LIN {X -0.125,Y -582.899,Z 496.268,A 0.000,B 0.000,C 90.000,E1 264.261} C_DIS
LIN {X -0.140,Y -579.949,Z 496.259,A 0.000,B 0.000,C 90.000,E1 262.648} C_DIS
LIN {X 0.066,Y -576.563,Z 496.249,A 0.000,B 0.000,C 90.000,E1 260.735} C_DIS
LIN {X -0.121,Y -574.110,Z 496.241,A 0.000,B 0.000,C 90.000,E1 259.398} C_DIS
LIN {X -0.046,Y -570.835,Z 496.232,A 0.000,B 0.000,C 90.000,E1 257.757} C_DIS
LIN {X -0.043,Y -567.459,Z 496.223,A 0.000,B 0.000,C 90.000,E1 256.117} C_DIS
LIN {X 0.233,Y -565.087,Z 496.217,A 0.000,B 0.000,C 90.000,E1 254.991} C_DIS
LIN {X -0.069,Y -562.642,Z 496.211,A 0.000,B 0.000,C 90.000,E1 253.921} C_DIS
LIN {X -0.106,Y -559.363,Z 496.203,A 0.000,B 0.000,C 90.000,E1 252.543} C_DIS
LIN {X -0.026,Y -555.962,Z 496.195,A 0.000,B 0.000,C 90.000,E1 251.148} C_DIS
LIN {X 0.080,Y -551.464,Z 496.186,A 0.000,B 0.000,C 90.000,E1 249.464} C_DIS
LIN {X 0.139,Y -548.336,Z 496.180,A 0.000,B 0.000,C 90.000,E1 248.337} C_DIS
LIN {X -0.042,Y -545.121,Z 496.174,A 0.000,B 0.000,C 90.000,E1 247.230} C_DIS
LIN {X -0.059,Y -541.722,Z 496.167,A 0.000,B 0.000,C 90.000,E1 246.102} C_DIS
LIN {X 0.095,Y -537.343,Z 496.159,A 0.000,B 0.000,C 90.000,E1 244.665} C_DIS
LIN {X 0.192,Y -533.762,Z 496.153,A 0.000,B 0.000,C 90.000,E1 243.512} C_DIS
LIN {X 0.238,Y -530.130,Z 496.147,A 0.000,B 0.000,C 90.000,E1 242.359} C_DIS
LIN {X 0.260,Y -523.726,Z 496.135,A 0.000,B 0.000,C 90.000,E1 240.333} C_DIS
LIN {X -0.110,Y -519.148,Z 496.127,A 0.000,B 0.000,C 90.000,E1 238.918} C_DIS
LIN {X -0.043,Y -515.453,Z 496.121,A 0.000,B 0.000,C 90.000,E1 237.740} C_DIS
LIN {X 0.053,Y -509.649,Z 496.111,A 0.000,B 0.000,C 90.000,E1 235.960} C_DIS
LIN {X -0.004,Y -504.726,Z 496.103,A 0.000,B 0.000,C 90.000,E1 234.482} C_DIS
LIN {X 0.032,Y -498.936,Z 496.093,A 0.000,B 0.000,C 90.000,E1 232.683} C_DIS
LIN {X -0.033,Y -489.905,Z 496.076,A 0.000,B 0.000,C 90.000,E1 229.666} C_DIS
LIN {X -0.260,Y -483.929,Z 496.064,A 0.000,B 0.000,C 90.000,E1 227.553} C_DIS
LIN {X 0.082,Y -479.810,Z 496.056,A 0.000,B 0.000,C 90.000,E1 225.972} C_DIS
LIN {X 0.215,Y -474.180,Z 496.043,A 0.000,B 0.000,C 90.000,E1 223.785} C_DIS
LIN {X 0.047,Y -470.290,Z 496.035,A 0.000,B 0.000,C 90.000,E1 222.243} C_DIS
LIN {X -0.124,Y -465.832,Z 496.024,A 0.000,B 0.000,C 90.000,E1 220.378} C_DIS
LIN {X -0.245,Y -460.903,Z 496.012,A 0.000,B 0.000,C 90.000,E1 218.177} C_DIS
LIN {X -0.034,Y -455.639,Z 495.998,A 0.000,B 0.000,C 90.000,E1 215.598} C_DIS
LIN {X 0.057,Y -451.793,Z 495.987,A 0.000,B 0.000,C 90.000,E1 213.658} C_DIS
LIN {X 0.051,Y -448.147,Z 495.976,A 0.000,B 0.000,C 90.000,E1 211.720} C_DIS
LIN {X -0.203,Y -445.158,Z 495.967,A 0.000,B 0.000,C 90.000,E1 210.129} C_DIS
LIN {X -0.235,Y -441.032,Z 495.955,A 0.000,B 0.000,C 90.000,E1 207.847} C_DIS
LIN {X -0.049,Y -438.068,Z 495.945,A 0.000,B 0.000,C 90.000,E1 206.181} C_DIS
LIN {X 0.060,Y -435.744,Z 495.938,A 0.000,B 0.000,C 90.000,E1 204.847} C_DIS
LIN {X -0.228,Y -432.280,Z 495.927,A 0.000,B 0.000,C 90.000,E1 202.898} C_DIS
LIN {X -0.159,Y -428.358,Z 495.914,A 0.000,B 0.000,C 90.000,E1 200.556} C_DIS
LIN {X -0.143,Y -425.321,Z 495.903,A 0.000,B 0.000,C 90.000,E1 198.544} C_DIS
LIN {X 0.128,Y -420.629,Z 495.884,A 0.000,B 0.000,C 90.000,E1 195.134} C_DIS
LIN {X 0.042,Y -417.671,Z 495.871,A 0.000,B 0.000,C 90.000,E1 192.771} C_DIS
LIN {X -0.001,Y -415.716,Z 495.862,A 0.000,B 0.000,C 90.000,E1 191.074} C_DIS
LIN {X -0.048,Y -413.433,Z 495.850,A 0.000,B 0.000,C 90.000,E1 189.029} C_DIS
LIN {X 0.132,Y -410.700,Z 495.835,A 0.000,B 0.000,C 90.000,E1 186.258} C_DIS
LIN {X 0.162,Y -408.347,Z 495.822,A 0.000,B 0.000,C 90.000,E1 183.841} C_DIS
LIN {X 0.002,Y -405.676,Z 495.802,A 0.000,B 0.000,C 90.000,E1 180.401} C_DIS
LIN {X 0.173,Y -403.932,Z 495.785,A 0.000,B 0.000,C 90.000,E1 177.249} C_DIS
LIN {X -0.065,Y -402.940,Z 495.766,A 0.000,B 0.000,C 90.000,E1 173.799} C_DIS
LIN {X -0.189,Y -402.803,Z 495.754,A 0.000,B 0.000,C 90.000,E1 171.724} C_DIS
LIN {X -0.134,Y -403.045,Z 495.738,A 0.000,B 0.000,C 90.000,E1 168.926} C_DIS
LIN {X 0.015,Y -403.828,Z 495.723,A 0.000,B 0.000,C 90.000,E1 166.117} C_DIS
LIN {X 0.083,Y -404.981,Z 495.707,A 0.000,B 0.000,C 90.000,E1 163.323} C_DIS
LIN {X 0.042,Y -406.645,Z 495.692,A 0.000,B 0.000,C 90.000,E1 160.550} C_DIS
LIN {X 0.212,Y -409.001,Z 495.675,A 0.000,B 0.000,C 90.000,E1 157.411} C_DIS
LIN {X 0.099,Y -410.828,Z 495.663,A 0.000,B 0.000,C 90.000,E1 155.357} C_DIS
LIN {X 0.000,Y -412.786,Z 495.652,A 0.000,B 0.000,C 90.000,E1 153.307} C_DIS
LIN {X 0.009,Y -414.381,Z 495.642,A 0.000,B 0.000,C 90.000,E1 151.591} C_DIS
LIN {X 0.073,Y -415.964,Z 495.633,A 0.000,B 0.000,C 90.000,E1 149.871} C_DIS
LIN {X -0.238,Y -417.734,Z 495.621,A 0.000,B 0.000,C 90.000,E1 147.867} C_DIS
LIN {X -0.200,Y -418.862,Z 495.614,A 0.000,B 0.000,C 90.000,E1 146.501} C_DIS
LIN {X 0.046,Y -420.250,Z 495.604,A 0.000,B 0.000,C 90.000,E1 144.769} C_DIS
LIN {X 0.054,Y -422.224,Z 495.591,A 0.000,B 0.000,C 90.000,E1 142.396} C_DIS
LIN {X 0.158,Y -423.798,Z 495.580,A 0.000,B 0.000,C 90.000,E1 140.356} C_DIS
LIN {X 0.115,Y -424.813,Z 495.572,A 0.000,B 0.000,C 90.000,E1 139.013} C_DIS
LIN {X 0.051,Y -425.666,Z 495.565,A 0.000,B 0.000,C 90.000,E1 137.676} C_DIS
LIN {X 0.093,Y -426.178,Z 495.559,A 0.000,B 0.000,C 90.000,E1 136.662} C_DIS
LIN {X 0.053,Y -426.740,Z 495.552,A 0.000,B 0.000,C 90.000,E1 135.324} C_DIS
LIN {X -0.285,Y -427.019,Z 495.544,A 0.000,B 0.000,C 90.000,E1 134.028} C_DIS
LIN {X 0.148,Y -427.105,Z 495.541,A 0.000,B 0.000,C 90.000,E1 133.299} C_DIS
LIN {X -0.085,Y -426.928,Z 495.535,A 0.000,B 0.000,C 90.000,E1 132.324} C_DIS
LIN {X -0.120,Y -426.340,Z 495.528,A 0.000,B 0.000,C 90.000,E1 130.987} C_DIS
LIN {X -0.029,Y -425.591,Z 495.522,A 0.000,B 0.000,C 90.000,E1 129.967} C_DIS
LIN {X -0.043,Y -424.318,Z 495.515,A 0.000,B 0.000,C 90.000,E1 128.624} C_DIS
LIN {X -0.088,Y -422.876,Z 495.507,A 0.000,B 0.000,C 90.000,E1 127.282} C_DIS
LIN {X -0.081,Y -421.282,Z 495.500,A 0.000,B 0.000,C 90.000,E1 125.931} C_DIS
LIN {X 0.004,Y -419.535,Z 495.492,A 0.000,B 0.000,C 90.000,E1 124.565} C_DIS
LIN {X -0.110,Y -419.290,Z 495.491,A 0.000,B 0.000,C 90.000,E1 124.405} C_DIS
LIN {X -0.148,Y -419.282,Z 495.491,A 0.000,B 0.000,C 90.000,E1 124.405} C_DIS
LIN {X 0.029,Y -429.026,Z 495.471,A 0.000,B 0.000,C 90.000,E1 120.846} C_DIS
LIN {X -0.198,Y -431.019,Z 495.468,A 0.000,B 0.000,C 90.000,E1 120.207} C_DIS
LIN {X -0.054,Y -440.094,Z 495.447,A 0.000,B 0.000,C 90.000,E1 116.539} C_DIS
LIN {X -0.056,Y -444.873,Z 495.438,A 0.000,B 0.000,C 90.000,E1 114.899} C_DIS
LIN {X 0.203,Y -453.984,Z 495.417,A 0.000,B 0.000,C 90.000,E1 110.972} C_DIS
LIN {X -0.270,Y -456.632,Z 495.411,A 0.000,B 0.000,C 90.000,E1 110.066} C_DIS
LIN {X 0.061,Y -457.448,Z 495.410,A 0.000,B 0.000,C 90.000,E1 109.704} C_DIS
LIN {X -0.005,Y -464.473,Z 495.390,A 0.000,B 0.000,C 90.000,E1 106.260} C_DIS
LIN {X -0.045,Y -464.485,Z 495.390,A 0.000,B 0.000,C 90.000,E1 106.260} C_DIS
LIN {X 0.015,Y -471.360,Z 495.390,A 0.000,B 0.000,C 90.000,E1 106.134} C_DIS
LIN {X -0.014,Y -475.196,Z 495.389,A 0.000,B 0.000,C 90.000,E1 106.079} C_DIS
LIN {X -0.202,Y -485.320,Z 495.388,A 0.000,B 0.000,C 90.000,E1 105.898} C_DIS
LIN {X 0.014,Y -492.601,Z 495.387,A 0.000,B 0.000,C 90.000,E1 105.717} C_DIS
LIN {X 0.107,Y -506.770,Z 495.385,A 0.000,B 0.000,C 90.000,E1 105.371} C_DIS
LIN {X -0.249,Y -517.096,Z 495.384,A 0.000,B 0.000,C 90.000,E1 105.134} C_DIS
LIN {X -0.215,Y -527.592,Z 495.382,A 0.000,B 0.000,C 90.000,E1 104.828} C_DIS
LIN {X 0.032,Y -537.871,Z 495.381,A 0.000,B 0.000,C 90.000,E1 104.481} C_DIS
LIN {X 0.104,Y -544.566,Z 495.379,A 0.000,B 0.000,C 90.000,E1 104.245} C_DIS
LIN {X -0.050,Y -551.197,Z 495.378,A 0.000,B 0.000,C 90.000,E1 104.008} C_DIS
LIN {X -0.155,Y -554.500,Z 495.377,A 0.000,B 0.000,C 90.000,E1 103.883} C_DIS
LIN {X 0.048,Y -564.165,Z 495.375,A 0.000,B 0.000,C 90.000,E1 103.411} C_DIS
LIN {X 0.216,Y -567.305,Z 495.374,A 0.000,B 0.000,C 90.000,E1 103.244} C_DIS
LIN {X -0.224,Y -576.586,Z 495.371,A 0.000,B 0.000,C 90.000,E1 102.771} C_DIS
LIN {X 0.092,Y -582.403,Z 495.369,A 0.000,B 0.000,C 90.000,E1 102.355} C_DIS
LIN {X 0.026,Y -586.631,Z 495.367,A 0.000,B 0.000,C 90.000,E1 102.063} C_DIS
LIN {X 0.092,Y -588.353,Z 495.366,A 0.000,B 0.000,C 90.000,E1 101.951} C_DIS
LIN {X 0.279,Y -596.480,Z 495.363,A 0.000,B 0.000,C 90.000,E1 101.299} C_DIS
LIN {X 0.316,Y -600.049,Z 495.361,A 0.000,B 0.000,C 90.000,E1 101.007} C_DIS
LIN {X 0.142,Y -606.738,Z 495.358,A 0.000,B 0.000,C 90.000,E1 100.433} C_DIS
LIN {X -0.193,Y -612.950,Z 495.355,A 0.000,B 0.000,C 90.000,E1 99.849} C_DIS
LIN {X 0.032,Y -617.750,Z 495.352,A 0.000,B 0.000,C 90.000,E1 99.321} C_DIS
LIN {X 0.023,Y -623.315,Z 495.348,A 0.000,B 0.000,C 90.000,E1 98.681} C_DIS
LIN {X 0.098,Y -627.427,Z 495.345,A 0.000,B 0.000,C 90.000,E1 98.163} C_DIS
LIN {X 0.060,Y -632.061,Z 495.342,A 0.000,B 0.000,C 90.000,E1 97.530} C_DIS
LIN {X 0.005,Y -636.964,Z 495.338,A 0.000,B 0.000,C 90.000,E1 96.777} C_DIS
LIN {X 0.180,Y -639.953,Z 495.335,A 0.000,B 0.000,C 90.000,E1 96.258} C_DIS
LIN {X 0.171,Y -644.017,Z 495.331,A 0.000,B 0.000,C 90.000,E1 95.511} C_DIS
LIN {X 0.103,Y -648.345,Z 495.326,A 0.000,B 0.000,C 90.000,E1 94.645} C_DIS
LIN {X 0.303,Y -650.663,Z 495.323,A 0.000,B 0.000,C 90.000,E1 94.131} C_DIS
LIN {X -0.296,Y -653.703,Z 495.319,A 0.000,B 0.000,C 90.000,E1 93.440} C_DIS
LIN {X -0.018,Y -655.493,Z 495.316,A 0.000,B 0.000,C 90.000,E1 92.922} C_DIS
LIN {X 0.240,Y -657.038,Z 495.314,A 0.000,B 0.000,C 90.000,E1 92.407} C_DIS
LIN {X -0.312,Y -658.803,Z 495.309,A 0.000,B 0.000,C 90.000,E1 91.718} C_DIS
LIN {X -0.028,Y -659.700,Z 495.307,A 0.000,B 0.000,C 90.000,E1 91.203} C_DIS
LIN {X 0.265,Y -660.274,Z 495.304,A 0.000,B 0.000,C 90.000,E1 90.688} C_DIS
LIN {X -0.275,Y -660.761,Z 495.300,A 0.000,B 0.000,C 90.000,E1 90.000} C_DIS
LIN {X 0.029,Y -660.764,Z 495.297,A 0.000,B 0.000,C 90.000,E1 89.484} C_DIS
LIN {X 0.151,Y -660.208,Z 495.293,A 0.000,B 0.000,C 90.000,E1 88.740} C_DIS
LIN {X -0.212,Y -659.627,Z 495.290,A 0.000,B 0.000,C 90.000,E1 88.282} C_DIS
LIN {X 0.103,Y -658.852,Z 495.288,A 0.000,B 0.000,C 90.000,E1 87.764} C_DIS
LIN {X -0.268,Y -657.826,Z 495.285,A 0.000,B 0.000,C 90.000,E1 87.306} C_DIS
LIN {X -0.148,Y -655.795,Z 495.281,A 0.000,B 0.000,C 90.000,E1 86.560} C_DIS
LIN {X 0.111,Y -654.200,Z 495.278,A 0.000,B 0.000,C 90.000,E1 86.045} C_DIS
LIN {X -0.249,Y -652.384,Z 495.275,A 0.000,B 0.000,C 90.000,E1 85.584} C_DIS
LIN {X 0.034,Y -650.350,Z 495.273,A 0.000,B 0.000,C 90.000,E1 85.065} C_DIS
LIN {X 0.081,Y -646.848,Z 495.269,A 0.000,B 0.000,C 90.000,E1 84.318} C_DIS
LIN {X 0.205,Y -643.584,Z 495.265,A 0.000,B 0.000,C 90.000,E1 83.685} C_DIS
LIN {X -0.339,Y -640.018,Z 495.262,A 0.000,B 0.000,C 90.000,E1 83.109} C_DIS
LIN {X -0.197,Y -636.089,Z 495.258,A 0.000,B 0.000,C 90.000,E1 82.470} C_DIS
LIN {X -0.169,Y -631.793,Z 495.255,A 0.000,B 0.000,C 90.000,E1 81.837} C_DIS
LIN {X -0.036,Y -628.041,Z 495.252,A 0.000,B 0.000,C 90.000,E1 81.319} C_DIS
LIN {X 0.054,Y -622.961,Z 495.248,A 0.000,B 0.000,C 90.000,E1 80.679} C_DIS
LIN {X 0.135,Y -617.609,Z 495.245,A 0.000,B 0.000,C 90.000,E1 80.038} C_DIS
LIN {X 0.094,Y -611.756,Z 495.241,A 0.000,B 0.000,C 90.000,E1 79.398} C_DIS
LIN {X 0.139,Y -605.468,Z 495.238,A 0.000,B 0.000,C 90.000,E1 78.757} C_DIS
LIN {X -0.032,Y -600.385,Z 495.235,A 0.000,B 0.000,C 90.000,E1 78.285} C_DIS
LIN {X -0.205,Y -596.393,Z 495.233,A 0.000,B 0.000,C 90.000,E1 77.937} C_DIS
LIN {X -0.068,Y -590.433,Z 495.230,A 0.000,B 0.000,C 90.000,E1 77.465} C_DIS
LIN {X 0.344,Y -584.507,Z 495.228,A 0.000,B 0.000,C 90.000,E1 76.992} C_DIS
LIN {X -0.283,Y -578.256,Z 495.226,A 0.000,B 0.000,C 90.000,E1 76.645} C_DIS
LIN {X -0.252,Y -573.325,Z 495.224,A 0.000,B 0.000,C 90.000,E1 76.353} C_DIS
LIN {X -0.124,Y -566.598,Z 495.222,A 0.000,B 0.000,C 90.000,E1 75.992} C_DIS
LIN {X -0.266,Y -559.098,Z 495.220,A 0.000,B 0.000,C 90.000,E1 75.700} C_DIS
LIN {X 0.117,Y -555.118,Z 495.220,A 0.000,B 0.000,C 90.000,E1 75.519} C_DIS
LIN {X 0.209,Y -547.325,Z 495.218,A 0.000,B 0.000,C 90.000,E1 75.283} C_DIS
LIN {X -0.047,Y -540.716,Z 495.218,A 0.000,B 0.000,C 90.000,E1 75.172} C_DIS
LIN {X 0.174,Y -534.917,Z 495.217,A 0.000,B 0.000,C 90.000,E1 75.046} C_DIS
LIN {X -0.132,Y -527.738,Z 495.217,A 0.000,B 0.000,C 90.000,E1 74.991} C_DIS
LIN {X -0.034,Y -523.125,Z 495.216,A 0.000,B 0.000,C 90.000,E1 74.936} C_DIS
LIN {X 0.189,Y -512.995,Z 495.216,A 0.000,B 0.000,C 90.000,E1 74.866} C_DIS
LIN {X -0.025,Y -504.486,Z 495.216,A 0.000,B 0.000,C 90.000,E1 74.866} C_DIS
LIN {X -0.053,Y -477.448,Z 495.216,A 0.000,B 0.000,C 90.000,E1 74.866} C_DIS
LIN {X 0.011,Y -474.312,Z 495.201,A 0.000,B 0.000,C 90.000,E1 72.236} C_DIS
LIN {X -0.168,Y -473.904,Z 495.200,A 0.000,B 0.000,C 90.000,E1 71.945} C_DIS
LIN {X -0.041,Y -466.293,Z 495.175,A 0.000,B 0.000,C 90.000,E1 67.539} C_DIS
LIN {X -0.099,Y -465.863,Z 495.173,A 0.000,B 0.000,C 90.000,E1 67.230} C_DIS
LIN {X -0.157,Y -465.298,Z 495.172,A 0.000,B 0.000,C 90.000,E1 66.922} C_DIS
LIN {X 0.220,Y -456.907,Z 495.149,A 0.000,B 0.000,C 90.000,E1 62.743} C_DIS
LIN {X -0.076,Y -455.278,Z 495.143,A 0.000,B 0.000,C 90.000,E1 61.820} C_DIS
LIN {X -0.221,Y -450.847,Z 495.133,A 0.000,B 0.000,C 90.000,E1 59.999} C_DIS
LIN {X 0.130,Y -450.870,Z 495.133,A 0.000,B 0.000,C 90.000,E1 59.950} C_DIS
LIN {X -0.043,Y -456.053,Z 495.127,A 0.000,B 0.000,C 90.000,E1 58.918} C_DIS
LIN {X 0.049,Y -460.472,Z 495.122,A 0.000,B 0.000,C 90.000,E1 57.946} C_DIS
LIN {X -0.097,Y -463.771,Z 495.118,A 0.000,B 0.000,C 90.000,E1 57.168} C_DIS
LIN {X -0.074,Y -466.800,Z 495.113,A 0.000,B 0.000,C 90.000,E1 56.373} C_DIS
LIN {X 0.091,Y -468.866,Z 495.110,A 0.000,B 0.000,C 90.000,E1 55.722} C_DIS
LIN {X 0.170,Y -471.543,Z 495.104,A 0.000,B 0.000,C 90.000,E1 54.769} C_DIS
LIN {X 0.166,Y -473.662,Z 495.099,A 0.000,B 0.000,C 90.000,E1 53.829} C_DIS
LIN {X 0.118,Y -474.920,Z 495.096,A 0.000,B 0.000,C 90.000,E1 53.210} C_DIS
LIN {X -0.052,Y -476.778,Z 495.089,A 0.000,B 0.000,C 90.000,E1 51.984} C_DIS
LIN {X -0.165,Y -477.602,Z 495.085,A 0.000,B 0.000,C 90.000,E1 51.376} C_DIS
LIN {X -0.098,Y -478.550,Z 495.080,A 0.000,B 0.000,C 90.000,E1 50.436} C_DIS
LIN {X 0.196,Y -479.882,Z 495.072,A 0.000,B 0.000,C 90.000,E1 48.852} C_DIS
LIN {X 0.031,Y -480.562,Z 495.065,A 0.000,B 0.000,C 90.000,E1 47.634} C_DIS
LIN {X 0.074,Y -480.980,Z 495.060,A 0.000,B 0.000,C 90.000,E1 46.701} C_DIS
LIN {X -0.227,Y -481.214,Z 495.054,A 0.000,B 0.000,C 90.000,E1 45.810} C_DIS
LIN {X -0.056,Y -481.357,Z 495.048,A 0.000,B 0.000,C 90.000,E1 44.555} C_DIS
LIN {X 0.120,Y -481.316,Z 495.041,A 0.000,B 0.000,C 90.000,E1 43.299} C_DIS
LIN {X -0.028,Y -480.996,Z 495.034,A 0.000,B 0.000,C 90.000,E1 42.081} C_DIS
LIN {X 0.142,Y -480.437,Z 495.027,A 0.000,B 0.000,C 90.000,E1 40.825} C_DIS
LIN {X -0.042,Y -479.466,Z 495.017,A 0.000,B 0.000,C 90.000,E1 38.991} C_DIS
LIN {X -0.241,Y -478.407,Z 495.006,A 0.000,B 0.000,C 90.000,E1 37.156} C_DIS
LIN {X -0.176,Y -477.402,Z 494.998,A 0.000,B 0.000,C 90.000,E1 35.598} C_DIS
LIN {X 0.050,Y -475.869,Z 494.987,A 0.000,B 0.000,C 90.000,E1 33.706} C_DIS
LIN {X -0.001,Y -474.826,Z 494.980,A 0.000,B 0.000,C 90.000,E1 32.467} C_DIS
LIN {X -0.141,Y -473.414,Z 494.972,A 0.000,B 0.000,C 90.000,E1 30.924} C_DIS
LIN {X 0.097,Y -471.814,Z 494.963,A 0.000,B 0.000,C 90.000,E1 29.333} C_DIS
LIN {X -0.090,Y -470.583,Z 494.956,A 0.000,B 0.000,C 90.000,E1 28.103} C_DIS
LIN {X -0.098,Y -468.318,Z 494.942,A 0.000,B 0.000,C 90.000,E1 25.591} C_DIS
LIN {X -0.275,Y -465.857,Z 494.925,A 0.000,B 0.000,C 90.000,E1 22.461} C_DIS
LIN {X 0.104,Y -464.382,Z 494.911,A 0.000,B 0.000,C 90.000,E1 19.885} C_DIS
LIN {X -0.021,Y -463.424,Z 494.900,A 0.000,B 0.000,C 90.000,E1 18.000} C_DIS
LIN {X -0.088,Y -462.455,Z 494.888,A 0.000,B 0.000,C 90.000,E1 15.788} C_DIS
LIN {X 0.070,Y -461.536,Z 494.870,A 0.000,B 0.000,C 90.000,E1 12.591} C_DIS
LIN {X -0.121,Y -461.260,Z 494.852,A 0.000,B 0.000,C 90.000,E1 9.434} C_DIS
LIN {X -0.130,Y -461.578,Z 494.838,A 0.000,B 0.000,C 90.000,E1 6.891} C_DIS
LIN {X -0.035,Y -462.931,Z 494.819,A 0.000,B 0.000,C 90.000,E1 3.383} C_DIS
LIN {X -0.139,Y -464.512,Z 494.805,A 0.000,B 0.000,C 90.000,E1 0.859} C_DIS
LIN {X 0.142,Y -466.475,Z 494.792,A 0.000,B 0.000,C 90.000,E1 358.511} C_DIS
LIN {X -0.081,Y -468.797,Z 494.780,A 0.000,B 0.000,C 90.000,E1 356.331} C_DIS
LIN {X -0.209,Y -471.421,Z 494.767,A 0.000,B 0.000,C 90.000,E1 354.147} C_DIS
LIN {X 0.180,Y -473.420,Z 494.759,A 0.000,B 0.000,C 90.000,E1 352.534} C_DIS
LIN {X -0.128,Y -476.341,Z 494.747,A 0.000,B 0.000,C 90.000,E1 350.387} C_DIS
LIN {X 0.200,Y -479.684,Z 494.734,A 0.000,B 0.000,C 90.000,E1 348.173} C_DIS
LIN {X 0.222,Y -484.142,Z 494.721,A 0.000,B 0.000,C 90.000,E1 345.700} C_DIS
LIN {X 0.157,Y -488.504,Z 494.709,A 0.000,B 0.000,C 90.000,E1 343.559} C_DIS
LIN {X -0.033,Y -491.770,Z 494.700,A 0.000,B 0.000,C 90.000,E1 342.054} C_DIS
LIN {X -0.070,Y -496.463,Z 494.689,A 0.000,B 0.000,C 90.000,E1 339.934} C_DIS
LIN {X 0.045,Y -499.848,Z 494.680,A 0.000,B 0.000,C 90.000,E1 338.411} C_DIS
LIN {X -0.061,Y -503.163,Z 494.672,A 0.000,B 0.000,C 90.000,E1 336.922} C_DIS
LIN {X 0.096,Y -506.347,Z 494.663,A 0.000,B 0.000,C 90.000,E1 335.409} C_DIS
LIN {X -0.142,Y -509.441,Z 494.655,A 0.000,B 0.000,C 90.000,E1 333.948} C_DIS
LIN {X 0.009,Y -513.160,Z 494.645,A 0.000,B 0.000,C 90.000,E1 332.153} C_DIS
LIN {X 0.136,Y -517.602,Z 494.634,A 0.000,B 0.000,C 90.000,E1 330.078} C_DIS
LIN {X 0.110,Y -522.861,Z 494.621,A 0.000,B 0.000,C 90.000,E1 327.740} C_DIS
LIN {X -0.038,Y -527.524,Z 494.610,A 0.000,B 0.000,C 90.000,E1 325.722} C_DIS
LIN {X -0.047,Y -531.597,Z 494.600,A 0.000,B 0.000,C 90.000,E1 323.989} C_DIS
LIN {X -0.093,Y -535.702,Z 494.590,A 0.000,B 0.000,C 90.000,E1 322.271} C_DIS
LIN {X 0.267,Y -539.018,Z 494.582,A 0.000,B 0.000,C 90.000,E1 320.803} C_DIS
LIN {X 0.275,Y -542.391,Z 494.575,A 0.000,B 0.000,C 90.000,E1 319.380} C_DIS
LIN {X -0.068,Y -545.702,Z 494.567,A 0.000,B 0.000,C 90.000,E1 318.000} C_DIS
LIN {X 0.018,Y -548.934,Z 494.559,A 0.000,B 0.000,C 90.000,E1 316.581} C_DIS
LIN {X 0.162,Y -552.044,Z 494.551,A 0.000,B 0.000,C 90.000,E1 315.162} C_DIS
LIN {X 0.016,Y -555.740,Z 494.542,A 0.000,B 0.000,C 90.000,E1 313.500} C_DIS
LIN {X -0.054,Y -559.395,Z 494.532,A 0.000,B 0.000,C 90.000,E1 311.838} C_DIS
LIN {X -0.103,Y -562.458,Z 494.525,A 0.000,B 0.000,C 90.000,E1 310.458} C_DIS
LIN {X -0.360,Y -566.015,Z 494.516,A 0.000,B 0.000,C 90.000,E1 308.830} C_DIS
LIN {X 0.029,Y -570.242,Z 494.505,A 0.000,B 0.000,C 90.000,E1 306.870} C_DIS
LIN {X 0.177,Y -574.605,Z 494.494,A 0.000,B 0.000,C 90.000,E1 304.945} C_DIS
LIN {X 0.265,Y -577.718,Z 494.487,A 0.000,B 0.000,C 90.000,E1 303.579} C_DIS
LIN {X -0.068,Y -582.051,Z 494.476,A 0.000,B 0.000,C 90.000,E1 301.720} C_DIS
LIN {X -0.161,Y -584.832,Z 494.469,A 0.000,B 0.000,C 90.000,E1 300.384} C_DIS
LIN {X 0.134,Y -586.980,Z 494.463,A 0.000,B 0.000,C 90.000,E1 299.283} C_DIS
LIN {X -0.048,Y -588.958,Z 494.457,A 0.000,B 0.000,C 90.000,E1 298.231} C_DIS
LIN {X -0.103,Y -590.292,Z 494.452,A 0.000,B 0.000,C 90.000,E1 297.436} C_DIS
LIN {X 0.004,Y -591.878,Z 494.447,A 0.000,B 0.000,C 90.000,E1 296.360} C_DIS
LIN {X 0.143,Y -593.252,Z 494.441,A 0.000,B 0.000,C 90.000,E1 295.283} C_DIS
LIN {X 0.302,Y -594.387,Z 494.435,A 0.000,B 0.000,C 90.000,E1 294.207} C_DIS
LIN {X -0.313,Y -595.281,Z 494.429,A 0.000,B 0.000,C 90.000,E1 293.206} C_DIS
LIN {X -0.004,Y -596.457,Z 494.420,A 0.000,B 0.000,C 90.000,E1 291.589} C_DIS
LIN {X -0.261,Y -597.158,Z 494.414,A 0.000,B 0.000,C 90.000,E1 290.556} C_DIS
LIN {X 0.263,Y -597.722,Z 494.408,A 0.000,B 0.000,C 90.000,E1 289.450} C_DIS
LIN {X -0.103,Y -598.445,Z 494.398,A 0.000,B 0.000,C 90.000,E1 287.638} C_DIS
LIN {X -0.225,Y -598.739,Z 494.394,A 0.000,B 0.000,C 90.000,E1 286.858} C_DIS
LIN {X 0.110,Y -599.251,Z 494.385,A 0.000,B 0.000,C 90.000,E1 285.245} C_DIS
LIN {X -0.003,Y -599.587,Z 494.377,A 0.000,B 0.000,C 90.000,E1 283.939} C_DIS
LIN {X -0.257,Y -599.822,Z 494.370,A 0.000,B 0.000,C 90.000,E1 282.647} C_DIS
LIN {X 0.078,Y -599.922,Z 494.363,A 0.000,B 0.000,C 90.000,E1 281.299} C_DIS
LIN {X 0.302,Y -599.890,Z 494.356,A 0.000,B 0.000,C 90.000,E1 279.962} C_DIS
LIN {X -0.070,Y -599.713,Z 494.348,A 0.000,B 0.000,C 90.000,E1 278.681} C_DIS
LIN {X 0.057,Y -599.361,Z 494.341,A 0.000,B 0.000,C 90.000,E1 277.352} C_DIS
LIN {X -0.111,Y -598.977,Z 494.335,A 0.000,B 0.000,C 90.000,E1 276.315} C_DIS
LIN {X -0.058,Y -598.209,Z 494.328,A 0.000,B 0.000,C 90.000,E1 274.992} C_DIS
LIN {X -0.019,Y -597.189,Z 494.320,A 0.000,B 0.000,C 90.000,E1 273.669} C_DIS
LIN {X -0.037,Y -596.002,Z 494.313,A 0.000,B 0.000,C 90.000,E1 272.350} C_DIS
LIN {X -0.078,Y -594.463,Z 494.306,A 0.000,B 0.000,C 90.000,E1 271.031} C_DIS
LIN {X -0.158,Y -592.713,Z 494.298,A 0.000,B 0.000,C 90.000,E1 269.714} C_DIS
LIN {X -0.273,Y -590.819,Z 494.291,A 0.000,B 0.000,C 90.000,E1 268.396} C_DIS
LIN {X -0.176,Y -588.465,Z 494.282,A 0.000,B 0.000,C 90.000,E1 266.788} C_DIS
LIN {X 0.237,Y -586.364,Z 494.275,A 0.000,B 0.000,C 90.000,E1 265.412} C_DIS
LIN {X -0.108,Y -584.532,Z 494.269,A 0.000,B 0.000,C 90.000,E1 264.375} C_DIS
LIN {X -0.312,Y -582.002,Z 494.261,A 0.000,B 0.000,C 90.000,E1 263.053} C_DIS
LIN {X 0.161,Y -579.504,Z 494.254,A 0.000,B 0.000,C 90.000,E1 261.659} C_DIS
LIN {X 0.148,Y -576.576,Z 494.245,A 0.000,B 0.000,C 90.000,E1 260.038} C_DIS
LIN {X -0.044,Y -573.904,Z 494.237,A 0.000,B 0.000,C 90.000,E1 258.701} C_DIS
LIN {X -0.172,Y -571.088,Z 494.230,A 0.000,B 0.000,C 90.000,E1 257.353} C_DIS
LIN {X -0.215,Y -568.227,Z 494.222,A 0.000,B 0.000,C 90.000,E1 255.992} C_DIS
LIN {X -0.138,Y -564.549,Z 494.213,A 0.000,B 0.000,C 90.000,E1 254.338} C_DIS
LIN {X -0.140,Y -561.268,Z 494.205,A 0.000,B 0.000,C 90.000,E1 252.960} C_DIS
LIN {X -0.202,Y -557.856,Z 494.198,A 0.000,B 0.000,C 90.000,E1 251.583} C_DIS
LIN {X 0.269,Y -554.949,Z 494.191,A 0.000,B 0.000,C 90.000,E1 250.423} C_DIS
LIN {X -0.015,Y -551.875,Z 494.185,A 0.000,B 0.000,C 90.000,E1 249.337} C_DIS
LIN {X -0.149,Y -548.743,Z 494.179,A 0.000,B 0.000,C 90.000,E1 248.230} C_DIS
LIN {X -0.119,Y -545.436,Z 494.173,A 0.000,B 0.000,C 90.000,E1 247.102} C_DIS
LIN {X 0.126,Y -542.890,Z 494.168,A 0.000,B 0.000,C 90.000,E1 246.230} C_DIS
LIN {X 0.077,Y -539.350,Z 494.162,A 0.000,B 0.000,C 90.000,E1 245.101} C_DIS
LIN {X -0.069,Y -534.880,Z 494.154,A 0.000,B 0.000,C 90.000,E1 243.691} C_DIS
LIN {X 0.181,Y -530.290,Z 494.146,A 0.000,B 0.000,C 90.000,E1 242.231} C_DIS
LIN {X 0.207,Y -523.855,Z 494.135,A 0.000,B 0.000,C 90.000,E1 240.205} C_DIS
LIN {X -0.164,Y -519.244,Z 494.127,A 0.000,B 0.000,C 90.000,E1 238.791} C_DIS
LIN {X 0.179,Y -515.530,Z 494.120,A 0.000,B 0.000,C 90.000,E1 237.582} C_DIS
LIN {X 0.284,Y -509.685,Z 494.110,A 0.000,B 0.000,C 90.000,E1 235.801} C_DIS
LIN {X -0.063,Y -504.725,Z 494.102,A 0.000,B 0.000,C 90.000,E1 234.356} C_DIS
LIN {X -0.033,Y -498.915,Z 494.092,A 0.000,B 0.000,C 90.000,E1 232.557} C_DIS
LIN {X 0.048,Y -490.779,Z 494.077,A 0.000,B 0.000,C 90.000,E1 229.828} C_DIS
LIN {X 0.019,Y -485.592,Z 494.067,A 0.000,B 0.000,C 90.000,E1 228.000} C_DIS
LIN {X 0.064,Y -481.441,Z 494.058,A 0.000,B 0.000,C 90.000,E1 226.458} C_DIS
LIN {X -0.322,Y -474.926,Z 494.044,A 0.000,B 0.000,C 90.000,E1 224.028} C_DIS
LIN {X -0.154,Y -471.027,Z 494.036,A 0.000,B 0.000,C 90.000,E1 222.447} C_DIS
LIN {X 0.041,Y -466.546,Z 494.025,A 0.000,B 0.000,C 90.000,E1 220.539} C_DIS
LIN {X -0.025,Y -460.911,Z 494.011,A 0.000,B 0.000,C 90.000,E1 218.016} C_DIS
LIN {X -0.192,Y -456.291,Z 493.999,A 0.000,B 0.000,C 90.000,E1 215.804} C_DIS
LIN {X 0.257,Y -451.820,Z 493.986,A 0.000,B 0.000,C 90.000,E1 213.499} C_DIS
LIN {X 0.005,Y -448.199,Z 493.976,A 0.000,B 0.000,C 90.000,E1 211.592} C_DIS
LIN {X -0.180,Y -444.608,Z 493.965,A 0.000,B 0.000,C 90.000,E1 209.667} C_DIS
LIN {X -0.228,Y -440.497,Z 493.952,A 0.000,B 0.000,C 90.000,E1 207.385} C_DIS
LIN {X -0.223,Y -436.977,Z 493.941,A 0.000,B 0.000,C 90.000,E1 205.412} C_DIS
LIN {X -0.087,Y -432.888,Z 493.928,A 0.000,B 0.000,C 90.000,E1 203.078} C_DIS
LIN {X -0.218,Y -429.444,Z 493.917,A 0.000,B 0.000,C 90.000,E1 201.099} C_DIS
LIN {X 0.020,Y -425.842,Z 493.904,A 0.000,B 0.000,C 90.000,E1 198.725} C_DIS
LIN {X -0.094,Y -421.065,Z 493.885,A 0.000,B 0.000,C 90.000,E1 195.371} C_DIS
LIN {X -0.168,Y -418.062,Z 493.872,A 0.000,B 0.000,C 90.000,E1 193.008} C_DIS
LIN {X -0.120,Y -416.080,Z 493.863,A 0.000,B 0.000,C 90.000,E1 191.299} C_DIS
LIN {X -0.189,Y -413.398,Z 493.849,A 0.000,B 0.000,C 90.000,E1 188.916} C_DIS
LIN {X -0.004,Y -410.661,Z 493.834,A 0.000,B 0.000,C 90.000,E1 186.144} C_DIS
LIN {X 0.017,Y -408.666,Z 493.823,A 0.000,B 0.000,C 90.000,E1 184.073} C_DIS
LIN {X -0.105,Y -405.932,Z 493.803,A 0.000,B 0.000,C 90.000,E1 180.630} C_DIS
LIN {X 0.044,Y -403.999,Z 493.784,A 0.000,B 0.000,C 90.000,E1 177.135} C_DIS
LIN {X 0.199,Y -402.989,Z 493.761,A 0.000,B 0.000,C 90.000,E1 172.932} C_DIS
LIN {X 0.132,Y -403.097,Z 493.742,A 0.000,B 0.000,C 90.000,E1 169.454} C_DIS
LIN {X -0.024,Y -404.024,Z 493.722,A 0.000,B 0.000,C 90.000,E1 165.992} C_DIS
LIN {X 0.060,Y -405.221,Z 493.707,A 0.000,B 0.000,C 90.000,E1 163.196} C_DIS
LIN {X 0.033,Y -406.934,Z 493.691,A 0.000,B 0.000,C 90.000,E1 160.423} C_DIS
LIN {X 0.061,Y -409.354,Z 493.674,A 0.000,B 0.000,C 90.000,E1 157.305} C_DIS
LIN {X 0.116,Y -411.217,Z 493.663,A 0.000,B 0.000,C 90.000,E1 155.229} C_DIS
LIN {X 0.028,Y -413.220,Z 493.651,A 0.000,B 0.000,C 90.000,E1 153.179} C_DIS
LIN {X 0.045,Y -414.830,Z 493.642,A 0.000,B 0.000,C 90.000,E1 151.463} C_DIS
LIN {X 0.117,Y -416.427,Z 493.632,A 0.000,B 0.000,C 90.000,E1 149.744} C_DIS
LIN {X 0.039,Y -418.287,Z 493.621,A 0.000,B 0.000,C 90.000,E1 147.709} C_DIS
LIN {X 0.049,Y -419.728,Z 493.611,A 0.000,B 0.000,C 90.000,E1 146.008} C_DIS
LIN {X -0.026,Y -421.164,Z 493.602,A 0.000,B 0.000,C 90.000,E1 144.322} C_DIS
LIN {X 0.016,Y -423.236,Z 493.589,A 0.000,B 0.000,C 90.000,E1 141.949} C_DIS
LIN {X -0.077,Y -424.597,Z 493.579,A 0.000,B 0.000,C 90.000,E1 140.275} C_DIS
LIN {X -0.106,Y -425.666,Z 493.572,A 0.000,B 0.000,C 90.000,E1 138.933} C_DIS
LIN {X 0.158,Y -426.570,Z 493.564,A 0.000,B 0.000,C 90.000,E1 137.553} C_DIS
LIN {X 0.122,Y -427.250,Z 493.557,A 0.000,B 0.000,C 90.000,E1 136.215} C_DIS
LIN {X -0.128,Y -427.675,Z 493.551,A 0.000,B 0.000,C 90.000,E1 135.243} C_DIS
LIN {X 0.232,Y -427.963,Z 493.546,A 0.000,B 0.000,C 90.000,E1 134.190} C_DIS
LIN {X -0.012,Y -428.111,Z 493.540,A 0.000,B 0.000,C 90.000,E1 133.218} C_DIS
LIN {X 0.055,Y -427.926,Z 493.535,A 0.000,B 0.000,C 90.000,E1 132.204} C_DIS
LIN {X 0.070,Y -427.366,Z 493.527,A 0.000,B 0.000,C 90.000,E1 130.862} C_DIS
LIN {X 0.084,Y -426.244,Z 493.520,A 0.000,B 0.000,C 90.000,E1 129.519} C_DIS
LIN {X 0.078,Y -424.934,Z 493.512,A 0.000,B 0.000,C 90.000,E1 128.177} C_DIS
LIN {X -0.217,Y -423.409,Z 493.505,A 0.000,B 0.000,C 90.000,E1 126.870} C_DIS
LIN {X 0.008,Y -421.233,Z 493.495,A 0.000,B 0.000,C 90.000,E1 125.152} C_DIS
LIN {X 0.052,Y -419.851,Z 493.490,A 0.000,B 0.000,C 90.000,E1 124.151} C_DIS
LIN {X 0.250,Y -419.858,Z 493.490,A 0.000,B 0.000,C 90.000,E1 124.119} C_DIS
LIN {X 0.112,Y -429.294,Z 493.471,A 0.000,B 0.000,C 90.000,E1 120.747} C_DIS
LIN {X 0.109,Y -430.332,Z 493.469,A 0.000,B 0.000,C 90.000,E1 120.413} C_DIS
LIN {X 0.109,Y -431.210,Z 493.467,A 0.000,B 0.000,C 90.000,E1 120.079} C_DIS
LIN {X 0.075,Y -440.334,Z 493.447,A 0.000,B 0.000,C 90.000,E1 116.437} C_DIS
LIN {X -0.168,Y -444.167,Z 493.440,A 0.000,B 0.000,C 90.000,E1 115.155} C_DIS
LIN {X -0.128,Y -445.054,Z 493.438,A 0.000,B 0.000,C 90.000,E1 114.823} C_DIS
LIN {X -0.038,Y -454.208,Z 493.416,A 0.000,B 0.000,C 90.000,E1 110.918} C_DIS
LIN {X 0.077,Y -456.869,Z 493.411,A 0.000,B 0.000,C 90.000,E1 109.939} C_DIS
LIN {X -0.020,Y -457.596,Z 493.409,A 0.000,B 0.000,C 90.000,E1 109.631} C_DIS
LIN {X -0.103,Y -465.482,Z 493.388,A 0.000,B 0.000,C 90.000,E1 105.843} C_DIS
LIN {X -0.143,Y -465.508,Z 493.388,A 0.000,B 0.000,C 90.000,E1 105.843} C_DIS
LIN {X 0.193,Y -478.092,Z 493.387,A 0.000,B 0.000,C 90.000,E1 105.607} C_DIS
LIN {X -0.069,Y -492.418,Z 493.385,A 0.000,B 0.000,C 90.000,E1 105.371} C_DIS
LIN {X -0.064,Y -506.458,Z 493.384,A 0.000,B 0.000,C 90.000,E1 105.064} C_DIS
LIN {X 0.216,Y -516.748,Z 493.382,A 0.000,B 0.000,C 90.000,E1 104.773} C_DIS
LIN {X -0.095,Y -530.722,Z 493.380,A 0.000,B 0.000,C 90.000,E1 104.411} C_DIS
LIN {X 0.173,Y -541.061,Z 493.378,A 0.000,B 0.000,C 90.000,E1 104.064} C_DIS
LIN {X 0.160,Y -547.737,Z 493.377,A 0.000,B 0.000,C 90.000,E1 103.828} C_DIS
LIN {X -0.063,Y -554.200,Z 493.376,A 0.000,B 0.000,C 90.000,E1 103.592} C_DIS
LIN {X -0.215,Y -564.012,Z 493.373,A 0.000,B 0.000,C 90.000,E1 103.175} C_DIS
LIN {X 0.167,Y -570.400,Z 493.371,A 0.000,B 0.000,C 90.000,E1 102.827} C_DIS
LIN {X 0.196,Y -576.510,Z 493.369,A 0.000,B 0.000,C 90.000,E1 102.479} C_DIS
LIN {X 0.203,Y -583.977,Z 493.367,A 0.000,B 0.000,C 90.000,E1 102.007} C_DIS
LIN {X 0.166,Y -588.497,Z 493.365,A 0.000,B 0.000,C 90.000,E1 101.715} C_DIS
LIN {X 0.175,Y -595.507,Z 493.362,A 0.000,B 0.000,C 90.000,E1 101.186} C_DIS
LIN {X -0.241,Y -599.770,Z 493.360,A 0.000,B 0.000,C 90.000,E1 100.894} C_DIS
LIN {X -0.085,Y -606.339,Z 493.357,A 0.000,B 0.000,C 90.000,E1 100.310} C_DIS
LIN {X 0.241,Y -611.470,Z 493.355,A 0.000,B 0.000,C 90.000,E1 99.792} C_DIS
LIN {X -0.300,Y -617.640,Z 493.351,A 0.000,B 0.000,C 90.000,E1 99.208} C_DIS
LIN {X 0.130,Y -623.031,Z 493.348,A 0.000,B 0.000,C 90.000,E1 98.568} C_DIS
LIN {X 0.204,Y -627.240,Z 493.345,A 0.000,B 0.000,C 90.000,E1 98.049} C_DIS
LIN {X 0.104,Y -632.809,Z 493.341,A 0.000,B 0.000,C 90.000,E1 97.296} C_DIS
LIN {X -0.021,Y -637.731,Z 493.336,A 0.000,B 0.000,C 90.000,E1 96.549} C_DIS
LIN {X -0.026,Y -642.064,Z 493.332,A 0.000,B 0.000,C 90.000,E1 95.796} C_DIS
LIN {X 0.182,Y -644.749,Z 493.329,A 0.000,B 0.000,C 90.000,E1 95.277} C_DIS
LIN {X 0.066,Y -649.038,Z 493.325,A 0.000,B 0.000,C 90.000,E1 94.416} C_DIS
LIN {X -0.160,Y -650.224,Z 493.323,A 0.000,B 0.000,C 90.000,E1 94.188} C_DIS
LIN {X -0.113,Y -653.277,Z 493.319,A 0.000,B 0.000,C 90.000,E1 93.440} C_DIS
LIN {X 0.163,Y -655.106,Z 493.316,A 0.000,B 0.000,C 90.000,E1 92.922} C_DIS
LIN {X -0.237,Y -656.619,Z 493.314,A 0.000,B 0.000,C 90.000,E1 92.465} C_DIS
LIN {X -0.137,Y -658.402,Z 493.310,A 0.000,B 0.000,C 90.000,E1 91.718} C_DIS
LIN {X 0.145,Y -659.308,Z 493.307,A 0.000,B 0.000,C 90.000,E1 91.203} C_DIS
LIN {X 0.254,Y -660.042,Z 493.303,A 0.000,B 0.000,C 90.000,E1 90.458} C_DIS
LIN {X -0.109,Y -660.323,Z 493.300,A 0.000,B 0.000,C 90.000,E1 90.000} C_DIS
LIN {X 0.192,Y -660.335,Z 493.297,A 0.000,B 0.000,C 90.000,E1 89.484} C_DIS
LIN {X 0.310,Y -659.755,Z 493.293,A 0.000,B 0.000,C 90.000,E1 88.740} C_DIS
LIN {X -0.055,Y -659.185,Z 493.290,A 0.000,B 0.000,C 90.000,E1 88.282} C_DIS
LIN {X 0.256,Y -658.356,Z 493.288,A 0.000,B 0.000,C 90.000,E1 87.764} C_DIS
LIN {X -0.118,Y -657.295,Z 493.285,A 0.000,B 0.000,C 90.000,E1 87.306} C_DIS
LIN {X 0.190,Y -655.952,Z 493.282,A 0.000,B 0.000,C 90.000,E1 86.788} C_DIS
LIN {X -0.202,Y -654.405,Z 493.280,A 0.000,B 0.000,C 90.000,E1 86.331} C_DIS
LIN {X 0.093,Y -652.644,Z 493.277,A 0.000,B 0.000,C 90.000,E1 85.812} C_DIS
LIN {X 0.164,Y -649.534,Z 493.273,A 0.000,B 0.000,C 90.000,E1 85.065} C_DIS
LIN {X 0.315,Y -646.569,Z 493.269,A 0.000,B 0.000,C 90.000,E1 84.432} C_DIS
LIN {X -0.083,Y -643.975,Z 493.267,A 0.000,B 0.000,C 90.000,E1 83.970} C_DIS
LIN {X 0.017,Y -640.399,Z 493.263,A 0.000,B 0.000,C 90.000,E1 83.337} C_DIS
LIN {X -0.242,Y -633.849,Z 493.257,A 0.000,B 0.000,C 90.000,E1 82.356} C_DIS
LIN {X 0.028,Y -628.587,Z 493.253,A 0.000,B 0.000,C 90.000,E1 81.602} C_DIS
LIN {X 0.123,Y -622.619,Z 493.249,A 0.000,B 0.000,C 90.000,E1 80.849} C_DIS
LIN {X 0.157,Y -617.069,Z 493.246,A 0.000,B 0.000,C 90.000,E1 80.208} C_DIS
LIN {X 0.187,Y -611.238,Z 493.242,A 0.000,B 0.000,C 90.000,E1 79.577} C_DIS
LIN {X -0.228,Y -606.216,Z 493.239,A 0.000,B 0.000,C 90.000,E1 79.106} C_DIS
LIN {X 0.062,Y -600.967,Z 493.237,A 0.000,B 0.000,C 90.000,E1 78.578} C_DIS
LIN {X -0.202,Y -595.407,Z 493.234,A 0.000,B 0.000,C 90.000,E1 78.117} C_DIS
LIN {X -0.081,Y -589.422,Z 493.231,A 0.000,B 0.000,C 90.000,E1 77.645} C_DIS
LIN {X -0.182,Y -583.249,Z 493.229,A 0.000,B 0.000,C 90.000,E1 77.229} C_DIS
LIN {X 0.242,Y -578.566,Z 493.227,A 0.000,B 0.000,C 90.000,E1 76.881} C_DIS
LIN {X 0.101,Y -571.843,Z 493.225,A 0.000,B 0.000,C 90.000,E1 76.520} C_DIS
LIN {X -0.085,Y -566.558,Z 493.224,A 0.000,B 0.000,C 90.000,E1 76.284} C_DIS
LIN {X -0.144,Y -559.264,Z 493.222,A 0.000,B 0.000,C 90.000,E1 75.992} C_DIS
LIN {X 0.264,Y -553.608,Z 493.221,A 0.000,B 0.000,C 90.000,E1 75.755} C_DIS
LIN {X -0.222,Y -547.880,Z 493.220,A 0.000,B 0.000,C 90.000,E1 75.644} C_DIS
LIN {X -0.104,Y -538.780,Z 493.219,A 0.000,B 0.000,C 90.000,E1 75.463} C_DIS
LIN {X -0.155,Y -534.537,Z 493.219,A 0.000,B 0.000,C 90.000,E1 75.408} C_DIS
LIN {X 0.171,Y -524.652,Z 493.218,A 0.000,B 0.000,C 90.000,E1 75.283} C_DIS
LIN {X -0.086,Y -519.148,Z 493.218,A 0.000,B 0.000,C 90.000,E1 75.283} C_DIS
LIN {X 0.182,Y -509.135,Z 493.218,A 0.000,B 0.000,C 90.000,E1 75.227} C_DIS
LIN {X 0.140,Y -477.998,Z 493.218,A 0.000,B 0.000,C 90.000,E1 75.227} C_DIS
LIN {X 0.038,Y -474.056,Z 493.200,A 0.000,B 0.000,C 90.000,E1 72.000} C_DIS
LIN {X 0.067,Y -465.488,Z 493.172,A 0.000,B 0.000,C 90.000,E1 66.975} C_DIS
LIN {X -0.153,Y -457.046,Z 493.149,A 0.000,B 0.000,C 90.000,E1 62.871} C_DIS
LIN {X -0.044,Y -455.461,Z 493.144,A 0.000,B 0.000,C 90.000,E1 61.897} C_DIS
LIN {X 0.251,Y -451.275,Z 493.134,A 0.000,B 0.000,C 90.000,E1 60.127} C_DIS
LIN {X 0.211,Y -451.285,Z 493.134,A 0.000,B 0.000,C 90.000,E1 60.127} C_DIS
LIN {X 0.023,Y -456.320,Z 493.129,A 0.000,B 0.000,C 90.000,E1 59.154} C_DIS
LIN {X -0.154,Y -459.421,Z 493.125,A 0.000,B 0.000,C 90.000,E1 58.535} C_DIS
LIN {X 0.078,Y -462.983,Z 493.121,A 0.000,B 0.000,C 90.000,E1 57.709} C_DIS
LIN {X -0.040,Y -465.626,Z 493.117,A 0.000,B 0.000,C 90.000,E1 57.089} C_DIS
LIN {X 0.252,Y -468.065,Z 493.114,A 0.000,B 0.000,C 90.000,E1 56.421} C_DIS
LIN {X 0.170,Y -470.149,Z 493.110,A 0.000,B 0.000,C 90.000,E1 55.801} C_DIS
LIN {X -0.124,Y -472.844,Z 493.105,A 0.000,B 0.000,C 90.000,E1 54.895} C_DIS
LIN {X -0.176,Y -474.326,Z 493.101,A 0.000,B 0.000,C 90.000,E1 54.276} C_DIS
LIN {X -0.148,Y -476.200,Z 493.096,A 0.000,B 0.000,C 90.000,E1 53.336} C_DIS
LIN {X -0.094,Y -477.639,Z 493.091,A 0.000,B 0.000,C 90.000,E1 52.396} C_DIS
LIN {X 0.176,Y -478.501,Z 493.088,A 0.000,B 0.000,C 90.000,E1 51.743} C_DIS
LIN {X 0.058,Y -479.744,Z 493.081,A 0.000,B 0.000,C 90.000,E1 50.517} C_DIS
LIN {X 0.010,Y -481.045,Z 493.072,A 0.000,B 0.000,C 90.000,E1 48.976} C_DIS
LIN {X -0.003,Y -481.833,Z 493.064,A 0.000,B 0.000,C 90.000,E1 47.433} C_DIS
LIN {X -0.071,Y -482.077,Z 493.060,A 0.000,B 0.000,C 90.000,E1 46.824} C_DIS
LIN {X -0.009,Y -482.291,Z 493.055,A 0.000,B 0.000,C 90.000,E1 45.891} C_DIS
LIN {X -0.159,Y -482.383,Z 493.048,A 0.000,B 0.000,C 90.000,E1 44.676} C_DIS
LIN {X 0.172,Y -482.270,Z 493.040,A 0.000,B 0.000,C 90.000,E1 43.095} C_DIS
LIN {X 0.008,Y -481.850,Z 493.033,A 0.000,B 0.000,C 90.000,E1 41.881} C_DIS
LIN {X 0.109,Y -481.407,Z 493.028,A 0.000,B 0.000,C 90.000,E1 40.943} C_DIS
LIN {X -0.110,Y -480.381,Z 493.017,A 0.000,B 0.000,C 90.000,E1 39.116} C_DIS
LIN {X 0.086,Y -479.315,Z 493.007,A 0.000,B 0.000,C 90.000,E1 37.237} C_DIS
LIN {X -0.021,Y -478.530,Z 493.000,A 0.000,B 0.000,C 90.000,E1 36.011} C_DIS
LIN {X 0.230,Y -477.029,Z 492.990,A 0.000,B 0.000,C 90.000,E1 34.119} C_DIS
LIN {X -0.015,Y -475.695,Z 492.981,A 0.000,B 0.000,C 90.000,E1 32.594} C_DIS
LIN {X -0.143,Y -474.255,Z 492.972,A 0.000,B 0.000,C 90.000,E1 31.052} C_DIS
LIN {X 0.110,Y -472.655,Z 492.964,A 0.000,B 0.000,C 90.000,E1 29.461} C_DIS
LIN {X 0.049,Y -470.778,Z 492.953,A 0.000,B 0.000,C 90.000,E1 27.590} C_DIS
LIN {X -0.103,Y -468.771,Z 492.941,A 0.000,B 0.000,C 90.000,E1 25.412} C_DIS
LIN {X -0.078,Y -466.297,Z 492.924,A 0.000,B 0.000,C 90.000,E1 22.259} C_DIS
LIN {X -0.232,Y -465.010,Z 492.911,A 0.000,B 0.000,C 90.000,E1 20.066} C_DIS
LIN {X 0.028,Y -463.892,Z 492.899,A 0.000,B 0.000,C 90.000,E1 17.819} C_DIS
LIN {X 0.181,Y -463.025,Z 492.888,A 0.000,B 0.000,C 90.000,E1 15.898} C_DIS
LIN {X -0.205,Y -462.013,Z 492.871,A 0.000,B 0.000,C 90.000,E1 12.771} C_DIS
LIN {X 0.087,Y -461.655,Z 492.853,A 0.000,B 0.000,C 90.000,E1 9.557} C_DIS
LIN {X 0.104,Y -461.897,Z 492.839,A 0.000,B 0.000,C 90.000,E1 7.011} C_DIS
LIN {X -0.201,Y -463.162,Z 492.820,A 0.000,B 0.000,C 90.000,E1 3.555} C_DIS
LIN {X 0.164,Y -464.696,Z 492.806,A 0.000,B 0.000,C 90.000,E1 0.974} C_DIS
LIN {X 0.147,Y -466.756,Z 492.792,A 0.000,B 0.000,C 90.000,E1 358.511} C_DIS
LIN {X -0.070,Y -469.047,Z 492.780,A 0.000,B 0.000,C 90.000,E1 356.331} C_DIS
LIN {X -0.192,Y -471.671,Z 492.767,A 0.000,B 0.000,C 90.000,E1 354.147} C_DIS
LIN {X 0.029,Y -474.101,Z 492.757,A 0.000,B 0.000,C 90.000,E1 352.243} C_DIS
LIN {X -0.098,Y -478.032,Z 492.741,A 0.000,B 0.000,C 90.000,E1 349.454} C_DIS
LIN {X -0.065,Y -483.830,Z 492.723,A 0.000,B 0.000,C 90.000,E1 346.047} C_DIS
LIN {X -0.266,Y -488.169,Z 492.711,A 0.000,B 0.000,C 90.000,E1 343.921} C_DIS
LIN {X 0.029,Y -492.106,Z 492.700,A 0.000,B 0.000,C 90.000,E1 342.054} C_DIS
LIN {X 0.002,Y -496.798,Z 492.689,A 0.000,B 0.000,C 90.000,E1 339.934} C_DIS
LIN {X 0.124,Y -500.215,Z 492.680,A 0.000,B 0.000,C 90.000,E1 338.411} C_DIS
LIN {X 0.024,Y -503.531,Z 492.672,A 0.000,B 0.000,C 90.000,E1 336.922} C_DIS
LIN {X 0.280,Y -507.399,Z 492.662,A 0.000,B 0.000,C 90.000,E1 335.101} C_DIS
LIN {X 0.156,Y -511.115,Z 492.652,A 0.000,B 0.000,C 90.000,E1 333.332} C_DIS
LIN {X -0.228,Y -514.249,Z 492.644,A 0.000,B 0.000,C 90.000,E1 331.897} C_DIS
LIN {X -0.188,Y -518.076,Z 492.634,A 0.000,B 0.000,C 90.000,E1 330.127} C_DIS
LIN {X -0.135,Y -522.754,Z 492.623,A 0.000,B 0.000,C 90.000,E1 328.074} C_DIS
LIN {X 0.119,Y -528.118,Z 492.610,A 0.000,B 0.000,C 90.000,E1 325.722} C_DIS
LIN {X 0.125,Y -532.240,Z 492.600,A 0.000,B 0.000,C 90.000,E1 323.989} C_DIS
LIN {X 0.095,Y -536.363,Z 492.590,A 0.000,B 0.000,C 90.000,E1 322.271} C_DIS
LIN {X -0.290,Y -539.721,Z 492.583,A 0.000,B 0.000,C 90.000,E1 320.884} C_DIS
LIN {X -0.276,Y -543.143,Z 492.575,A 0.000,B 0.000,C 90.000,E1 319.461} C_DIS
LIN {X 0.163,Y -546.491,Z 492.567,A 0.000,B 0.000,C 90.000,E1 318.000} C_DIS
LIN {X 0.299,Y -550.396,Z 492.557,A 0.000,B 0.000,C 90.000,E1 316.296} C_DIS
LIN {X -0.282,Y -554.123,Z 492.548,A 0.000,B 0.000,C 90.000,E1 314.676} C_DIS
LIN {X -0.006,Y -557.822,Z 492.539,A 0.000,B 0.000,C 90.000,E1 312.975} C_DIS
LIN {X -0.003,Y -561.539,Z 492.530,A 0.000,B 0.000,C 90.000,E1 311.310} C_DIS
LIN {X -0.014,Y -564.578,Z 492.522,A 0.000,B 0.000,C 90.000,E1 309.930} C_DIS
LIN {X 0.098,Y -567.560,Z 492.514,A 0.000,B 0.000,C 90.000,E1 308.543} C_DIS
LIN {X -0.059,Y -571.226,Z 492.505,A 0.000,B 0.000,C 90.000,E1 306.916} C_DIS
LIN {X -0.226,Y -575.642,Z 492.495,A 0.000,B 0.000,C 90.000,E1 305.025} C_DIS
LIN {X -0.120,Y -578.813,Z 492.487,A 0.000,B 0.000,C 90.000,E1 303.658} C_DIS
LIN {X 0.052,Y -581.900,Z 492.479,A 0.000,B 0.000,C 90.000,E1 302.291} C_DIS
LIN {X 0.239,Y -583.801,Z 492.475,A 0.000,B 0.000,C 90.000,E1 301.465} C_DIS
LIN {X 0.059,Y -587.101,Z 492.466,A 0.000,B 0.000,C 90.000,E1 299.873} C_DIS
LIN {X -0.233,Y -589.668,Z 492.459,A 0.000,B 0.000,C 90.000,E1 298.565} C_DIS
LIN {X 0.142,Y -591.490,Z 492.453,A 0.000,B 0.000,C 90.000,E1 297.462} C_DIS
LIN {X 0.011,Y -593.097,Z 492.447,A 0.000,B 0.000,C 90.000,E1 296.411} C_DIS
LIN {X 0.162,Y -594.524,Z 492.441,A 0.000,B 0.000,C 90.000,E1 295.335} C_DIS
LIN {X 0.089,Y -595.679,Z 492.435,A 0.000,B 0.000,C 90.000,E1 294.283} C_DIS
LIN {X 0.280,Y -596.613,Z 492.429,A 0.000,B 0.000,C 90.000,E1 293.206} C_DIS
LIN {X -0.157,Y -597.846,Z 492.420,A 0.000,B 0.000,C 90.000,E1 291.663} C_DIS
LIN {X -0.178,Y -598.585,Z 492.414,A 0.000,B 0.000,C 90.000,E1 290.610} C_DIS
LIN {X 0.162,Y -599.204,Z 492.409,A 0.000,B 0.000,C 90.000,E1 289.523} C_DIS
LIN {X 0.025,Y -600.003,Z 492.398,A 0.000,B 0.000,C 90.000,E1 287.692} C_DIS
LIN {X 0.207,Y -600.416,Z 492.393,A 0.000,B 0.000,C 90.000,E1 286.622} C_DIS
LIN {X 0.123,Y -600.927,Z 492.385,A 0.000,B 0.000,C 90.000,E1 285.315} C_DIS
LIN {X 0.048,Y -601.339,Z 492.378,A 0.000,B 0.000,C 90.000,E1 284.008} C_DIS
LIN {X -0.034,Y -601.595,Z 492.371,A 0.000,B 0.000,C 90.000,E1 282.703} C_DIS
LIN {X -0.099,Y -601.740,Z 492.365,A 0.000,B 0.000,C 90.000,E1 281.658} C_DIS
LIN {X 0.273,Y -601.784,Z 492.357,A 0.000,B 0.000,C 90.000,E1 280.310} C_DIS
LIN {X -0.065,Y -601.645,Z 492.350,A 0.000,B 0.000,C 90.000,E1 279.029} C_DIS
LIN {X 0.097,Y -601.355,Z 492.343,A 0.000,B 0.000,C 90.000,E1 277.701} C_DIS
LIN {X 0.255,Y -600.875,Z 492.336,A 0.000,B 0.000,C 90.000,E1 276.372} C_DIS
LIN {X -0.259,Y -600.126,Z 492.328,A 0.000,B 0.000,C 90.000,E1 275.106} C_DIS
LIN {X -0.189,Y -599.110,Z 492.321,A 0.000,B 0.000,C 90.000,E1 273.784} C_DIS
LIN {X -0.175,Y -597.900,Z 492.314,A 0.000,B 0.000,C 90.000,E1 272.465} C_DIS
LIN {X -0.184,Y -596.324,Z 492.306,A 0.000,B 0.000,C 90.000,E1 271.146} C_DIS
LIN {X -0.233,Y -594.572,Z 492.299,A 0.000,B 0.000,C 90.000,E1 269.828} C_DIS
LIN {X 0.278,Y -592.650,Z 492.292,A 0.000,B 0.000,C 90.000,E1 268.453} C_DIS
LIN {X -0.211,Y -590.238,Z 492.283,A 0.000,B 0.000,C 90.000,E1 266.906} C_DIS
LIN {X 0.268,Y -588.067,Z 492.275,A 0.000,B 0.000,C 90.000,E1 265.527} C_DIS
LIN {X -0.053,Y -586.188,Z 492.269,A 0.000,B 0.000,C 90.000,E1 264.489} C_DIS
LIN {X -0.226,Y -583.642,Z 492.262,A 0.000,B 0.000,C 90.000,E1 263.166} C_DIS
LIN {X -0.153,Y -580.574,Z 492.253,A 0.000,B 0.000,C 90.000,E1 261.546} C_DIS
LIN {X 0.302,Y -578.066,Z 492.246,A 0.000,B 0.000,C 90.000,E1 260.151} C_DIS
LIN {X 0.140,Y -575.362,Z 492.238,A 0.000,B 0.000,C 90.000,E1 258.814} C_DIS
LIN {X 0.240,Y -571.883,Z 492.229,A 0.000,B 0.000,C 90.000,E1 257.173} C_DIS
LIN {X -0.109,Y -569.577,Z 492.223,A 0.000,B 0.000,C 90.000,E1 256.117} C_DIS
LIN {X 0.140,Y -565.827,Z 492.214,A 0.000,B 0.000,C 90.000,E1 254.448} C_DIS
LIN {X 0.002,Y -562.524,Z 492.206,A 0.000,B 0.000,C 90.000,E1 253.087} C_DIS
LIN {X 0.133,Y -559.085,Z 492.198,A 0.000,B 0.000,C 90.000,E1 251.692} C_DIS
LIN {X 0.146,Y -556.932,Z 492.194,A 0.000,B 0.000,C 90.000,E1 250.859} C_DIS
LIN {X 0.173,Y -553.097,Z 492.186,A 0.000,B 0.000,C 90.000,E1 249.464} C_DIS
LIN {X -0.190,Y -549.152,Z 492.178,A 0.000,B 0.000,C 90.000,E1 248.103} C_DIS
LIN {X -0.148,Y -544.077,Z 492.169,A 0.000,B 0.000,C 90.000,E1 246.410} C_DIS
LIN {X -0.175,Y -540.520,Z 492.163,A 0.000,B 0.000,C 90.000,E1 245.281} C_DIS
LIN {X -0.048,Y -536.012,Z 492.155,A 0.000,B 0.000,C 90.000,E1 243.845} C_DIS
LIN {X -0.014,Y -531.380,Z 492.147,A 0.000,B 0.000,C 90.000,E1 242.410} C_DIS
LIN {X 0.102,Y -525.823,Z 492.137,A 0.000,B 0.000,C 90.000,E1 240.667} C_DIS
LIN {X 0.214,Y -521.219,Z 492.129,A 0.000,B 0.000,C 90.000,E1 239.203} C_DIS
LIN {X 0.167,Y -515.628,Z 492.119,A 0.000,B 0.000,C 90.000,E1 237.454} C_DIS
LIN {X 0.014,Y -511.721,Z 492.113,A 0.000,B 0.000,C 90.000,E1 236.294} C_DIS
LIN {X -0.096,Y -505.769,Z 492.103,A 0.000,B 0.000,C 90.000,E1 234.529} C_DIS
LIN {X -0.054,Y -498.924,Z 492.091,A 0.000,B 0.000,C 90.000,E1 232.431} C_DIS
LIN {X 0.170,Y -491.690,Z 492.078,A 0.000,B 0.000,C 90.000,E1 229.989} C_DIS
LIN {X 0.157,Y -486.464,Z 492.068,A 0.000,B 0.000,C 90.000,E1 228.162} C_DIS
LIN {X 0.001,Y -481.436,Z 492.057,A 0.000,B 0.000,C 90.000,E1 226.338} C_DIS
LIN {X -0.149,Y -475.711,Z 492.045,A 0.000,B 0.000,C 90.000,E1 224.190} C_DIS
LIN {X 0.124,Y -471.018,Z 492.035,A 0.000,B 0.000,C 90.000,E1 222.285} C_DIS
LIN {X -0.107,Y -467.300,Z 492.026,A 0.000,B 0.000,C 90.000,E1 220.744} C_DIS
LIN {X -0.194,Y -462.288,Z 492.014,A 0.000,B 0.000,C 90.000,E1 218.543} C_DIS
LIN {X -0.043,Y -457.622,Z 492.002,A 0.000,B 0.000,C 90.000,E1 216.297} C_DIS
LIN {X 0.068,Y -453.148,Z 491.989,A 0.000,B 0.000,C 90.000,E1 214.040} C_DIS
LIN {X -0.073,Y -448.856,Z 491.977,A 0.000,B 0.000,C 90.000,E1 211.799} C_DIS
LIN {X -0.085,Y -445.875,Z 491.968,A 0.000,B 0.000,C 90.000,E1 210.178} C_DIS
LIN {X -0.157,Y -442.315,Z 491.957,A 0.000,B 0.000,C 90.000,E1 208.231} C_DIS
LIN {X 0.053,Y -439.398,Z 491.948,A 0.000,B 0.000,C 90.000,E1 206.565} C_DIS
LIN {X 0.202,Y -436.429,Z 491.939,A 0.000,B 0.000,C 90.000,E1 204.899} C_DIS
LIN {X -0.076,Y -432.929,Z 491.927,A 0.000,B 0.000,C 90.000,E1 202.950} C_DIS
LIN {X 0.003,Y -428.951,Z 491.915,A 0.000,B 0.000,C 90.000,E1 200.610} C_DIS
LIN {X 0.025,Y -425.866,Z 491.903,A 0.000,B 0.000,C 90.000,E1 198.598} C_DIS
LIN {X 0.134,Y -421.524,Z 491.887,A 0.000,B 0.000,C 90.000,E1 195.552} C_DIS
LIN {X 0.169,Y -418.478,Z 491.873,A 0.000,B 0.000,C 90.000,E1 193.175} C_DIS
LIN {X 0.188,Y -416.065,Z 491.862,A 0.000,B 0.000,C 90.000,E1 191.130} C_DIS
LIN {X 0.036,Y -414.127,Z 491.853,A 0.000,B 0.000,C 90.000,E1 189.443} C_DIS
LIN {X -0.106,Y -411.317,Z 491.837,A 0.000,B 0.000,C 90.000,E1 186.720} C_DIS
LIN {X -0.036,Y -409.329,Z 491.826,A 0.000,B 0.000,C 90.000,E1 184.645} C_DIS
LIN {X -0.124,Y -406.689,Z 491.809,A 0.000,B 0.000,C 90.000,E1 181.547} C_DIS
LIN {X 0.127,Y -405.086,Z 491.795,A 0.000,B 0.000,C 90.000,E1 179.083} C_DIS
LIN {X -0.081,Y -403.811,Z 491.780,A 0.000,B 0.000,C 90.000,E1 176.331} C_DIS
LIN {X 0.120,Y -403.078,Z 491.760,A 0.000,B 0.000,C 90.000,E1 172.818} C_DIS
LIN {X 0.049,Y -403.247,Z 491.741,A 0.000,B 0.000,C 90.000,E1 169.342} C_DIS
LIN {X -0.105,Y -404.101,Z 491.723,A 0.000,B 0.000,C 90.000,E1 166.228} C_DIS
LIN {X -0.018,Y -405.297,Z 491.708,A 0.000,B 0.000,C 90.000,E1 163.433} C_DIS
LIN {X -0.172,Y -406.987,Z 491.693,A 0.000,B 0.000,C 90.000,E1 160.678} C_DIS
LIN {X -0.112,Y -409.103,Z 491.677,A 0.000,B 0.000,C 90.000,E1 157.901} C_DIS
LIN {X 0.157,Y -410.966,Z 491.666,A 0.000,B 0.000,C 90.000,E1 155.793} C_DIS
LIN {X 0.179,Y -413.302,Z 491.652,A 0.000,B 0.000,C 90.000,E1 153.384} C_DIS
LIN {X 0.027,Y -414.995,Z 491.643,A 0.000,B 0.000,C 90.000,E1 151.691} C_DIS
LIN {X -0.093,Y -416.623,Z 491.633,A 0.000,B 0.000,C 90.000,E1 149.999} C_DIS
LIN {X -0.032,Y -418.509,Z 491.622,A 0.000,B 0.000,C 90.000,E1 147.946} C_DIS
LIN {X 0.015,Y -419.721,Z 491.614,A 0.000,B 0.000,C 90.000,E1 146.580} C_DIS
LIN {X -0.107,Y -421.524,Z 491.603,A 0.000,B 0.000,C 90.000,E1 144.562} C_DIS
LIN {X -0.067,Y -423.622,Z 491.590,A 0.000,B 0.000,C 90.000,E1 142.190} C_DIS
LIN {X -0.155,Y -425.129,Z 491.581,A 0.000,B 0.000,C 90.000,E1 140.517} C_DIS
LIN {X 0.099,Y -426.235,Z 491.573,A 0.000,B 0.000,C 90.000,E1 139.138} C_DIS
LIN {X 0.003,Y -427.459,Z 491.564,A 0.000,B 0.000,C 90.000,E1 137.472} C_DIS
LIN {X -0.018,Y -428.201,Z 491.556,A 0.000,B 0.000,C 90.000,E1 136.134} C_DIS
LIN {X -0.178,Y -428.561,Z 491.553,A 0.000,B 0.000,C 90.000,E1 135.486} C_DIS
LIN {X 0.116,Y -428.970,Z 491.545,A 0.000,B 0.000,C 90.000,E1 134.109} C_DIS
LIN {X -0.118,Y -429.153,Z 491.540,A 0.000,B 0.000,C 90.000,E1 133.137} C_DIS
LIN {X 0.199,Y -428.863,Z 491.532,A 0.000,B 0.000,C 90.000,E1 131.757} C_DIS
LIN {X -0.008,Y -428.408,Z 491.527,A 0.000,B 0.000,C 90.000,E1 130.782} C_DIS
LIN {X 0.022,Y -427.300,Z 491.519,A 0.000,B 0.000,C 90.000,E1 129.439} C_DIS
LIN {X 0.031,Y -425.966,Z 491.512,A 0.000,B 0.000,C 90.000,E1 128.096} C_DIS
LIN {X 0.090,Y -424.346,Z 491.504,A 0.000,B 0.000,C 90.000,E1 126.744} C_DIS
LIN {X -0.251,Y -422.078,Z 491.495,A 0.000,B 0.000,C 90.000,E1 125.105} C_DIS
LIN {X 0.086,Y -420.447,Z 491.489,A 0.000,B 0.000,C 90.000,E1 123.913} C_DIS
LIN {X 0.047,Y -420.448,Z 491.488,A 0.000,B 0.000,C 90.000,E1 123.913} C_DIS
LIN {X 0.107,Y -430.579,Z 491.469,A 0.000,B 0.000,C 90.000,E1 120.335} C_DIS
LIN {X -0.092,Y -441.488,Z 491.445,A 0.000,B 0.000,C 90.000,E1 116.052} C_DIS
LIN {X -0.174,Y -444.401,Z 491.439,A 0.000,B 0.000,C 90.000,E1 115.079} C_DIS
LIN {X 0.084,Y -445.211,Z 491.437,A 0.000,B 0.000,C 90.000,E1 114.719} C_DIS
LIN {X -0.053,Y -454.411,Z 491.416,A 0.000,B 0.000,C 90.000,E1 110.844} C_DIS
LIN {X -0.094,Y -457.084,Z 491.410,A 0.000,B 0.000,C 90.000,E1 109.885} C_DIS
LIN {X 0.124,Y -462.803,Z 491.395,A 0.000,B 0.000,C 90.000,E1 106.985} C_DIS
LIN {X 0.119,Y -466.562,Z 491.386,A 0.000,B 0.000,C 90.000,E1 105.371} C_DIS
LIN {X 0.089,Y -466.765,Z 491.385,A 0.000,B 0.000,C 90.000,E1 105.371} C_DIS
LIN {X -0.008,Y -473.911,Z 491.385,A 0.000,B 0.000,C 90.000,E1 105.300} C_DIS
LIN {X 0.168,Y -486.273,Z 491.384,A 0.000,B 0.000,C 90.000,E1 105.079} C_DIS
LIN {X -0.034,Y -500.758,Z 491.382,A 0.000,B 0.000,C 90.000,E1 104.828} C_DIS
LIN {X 0.164,Y -507.675,Z 491.382,A 0.000,B 0.000,C 90.000,E1 104.662} C_DIS
LIN {X -0.014,Y -517.973,Z 491.380,A 0.000,B 0.000,C 90.000,E1 104.426} C_DIS
LIN {X -0.208,Y -532.009,Z 491.378,A 0.000,B 0.000,C 90.000,E1 104.064} C_DIS
LIN {X 0.111,Y -542.332,Z 491.376,A 0.000,B 0.000,C 90.000,E1 103.716} C_DIS
LIN {X 0.218,Y -548.839,Z 491.375,A 0.000,B 0.000,C 90.000,E1 103.480} C_DIS
LIN {X 0.025,Y -555.408,Z 491.374,A 0.000,B 0.000,C 90.000,E1 103.244} C_DIS
LIN {X 0.078,Y -563.708,Z 491.372,A 0.000,B 0.000,C 90.000,E1 102.883} C_DIS
LIN {X 0.215,Y -571.746,Z 491.370,A 0.000,B 0.000,C 90.000,E1 102.479} C_DIS
LIN {X -0.203,Y -574.860,Z 491.369,A 0.000,B 0.000,C 90.000,E1 102.355} C_DIS
LIN {X 0.172,Y -584.055,Z 491.366,A 0.000,B 0.000,C 90.000,E1 101.771} C_DIS
LIN {X 0.154,Y -588.528,Z 491.364,A 0.000,B 0.000,C 90.000,E1 101.478} C_DIS
LIN {X 0.056,Y -594.292,Z 491.362,A 0.000,B 0.000,C 90.000,E1 101.074} C_DIS
LIN {X -0.289,Y -597.789,Z 491.360,A 0.000,B 0.000,C 90.000,E1 100.838} C_DIS
LIN {X -0.140,Y -599.376,Z 491.359,A 0.000,B 0.000,C 90.000,E1 100.715} C_DIS
LIN {X 0.316,Y -607.053,Z 491.356,A 0.000,B 0.000,C 90.000,E1 100.018} C_DIS
LIN {X 0.173,Y -611.041,Z 491.354,A 0.000,B 0.000,C 90.000,E1 99.670} C_DIS
LIN {X -0.008,Y -615.898,Z 491.351,A 0.000,B 0.000,C 90.000,E1 99.208} C_DIS
LIN {X -0.234,Y -621.637,Z 491.348,A 0.000,B 0.000,C 90.000,E1 98.624} C_DIS
LIN {X 0.247,Y -628.005,Z 491.344,A 0.000,B 0.000,C 90.000,E1 97.814} C_DIS
LIN {X 0.214,Y -632.725,Z 491.340,A 0.000,B 0.000,C 90.000,E1 97.182} C_DIS
LIN {X 0.163,Y -637.714,Z 491.336,A 0.000,B 0.000,C 90.000,E1 96.429} C_DIS
LIN {X 0.214,Y -641.407,Z 491.332,A 0.000,B 0.000,C 90.000,E1 95.796} C_DIS
LIN {X 0.299,Y -644.788,Z 491.329,A 0.000,B 0.000,C 90.000,E1 95.163} C_DIS
LIN {X 0.184,Y -649.084,Z 491.324,A 0.000,B 0.000,C 90.000,E1 94.302} C_DIS
LIN {X -0.321,Y -651.788,Z 491.321,A 0.000,B 0.000,C 90.000,E1 93.726} C_DIS
LIN {X -0.265,Y -654.643,Z 491.316,A 0.000,B 0.000,C 90.000,E1 92.980} C_DIS
LIN {X -0.014,Y -656.139,Z 491.314,A 0.000,B 0.000,C 90.000,E1 92.465} C_DIS
LIN {X 0.082,Y -657.951,Z 491.310,A 0.000,B 0.000,C 90.000,E1 91.718} C_DIS
LIN {X -0.298,Y -658.866,Z 491.307,A 0.000,B 0.000,C 90.000,E1 91.260} C_DIS
LIN {X -0.194,Y -659.596,Z 491.303,A 0.000,B 0.000,C 90.000,E1 90.516} C_DIS
LIN {X 0.101,Y -659.867,Z 491.300,A 0.000,B 0.000,C 90.000,E1 90.000} C_DIS
LIN {X -0.261,Y -659.886,Z 491.297,A 0.000,B 0.000,C 90.000,E1 89.542} C_DIS
LIN {X -0.147,Y -659.293,Z 491.293,A 0.000,B 0.000,C 90.000,E1 88.797} C_DIS
LIN {X 0.143,Y -658.737,Z 491.291,A 0.000,B 0.000,C 90.000,E1 88.282} C_DIS
LIN {X -0.205,Y -657.862,Z 491.288,A 0.000,B 0.000,C 90.000,E1 87.822} C_DIS
LIN {X 0.074,Y -656.779,Z 491.285,A 0.000,B 0.000,C 90.000,E1 87.306} C_DIS
LIN {X 0.183,Y -654.632,Z 491.281,A 0.000,B 0.000,C 90.000,E1 86.560} C_DIS
LIN {X -0.218,Y -652.900,Z 491.278,A 0.000,B 0.000,C 90.000,E1 86.102} C_DIS
LIN {X -0.149,Y -649.868,Z 491.274,A 0.000,B 0.000,C 90.000,E1 85.355} C_DIS
LIN {X 0.003,Y -646.968,Z 491.271,A 0.000,B 0.000,C 90.000,E1 84.723} C_DIS
LIN {X 0.126,Y -643.674,Z 491.267,A 0.000,B 0.000,C 90.000,E1 84.090} C_DIS
LIN {X 0.217,Y -640.018,Z 491.264,A 0.000,B 0.000,C 90.000,E1 83.457} C_DIS
LIN {X -0.148,Y -636.693,Z 491.261,A 0.000,B 0.000,C 90.000,E1 82.989} C_DIS
LIN {X 0.212,Y -633.430,Z 491.258,A 0.000,B 0.000,C 90.000,E1 82.470} C_DIS
LIN {X 0.066,Y -627.843,Z 491.254,A 0.000,B 0.000,C 90.000,E1 81.724} C_DIS
LIN {X -0.051,Y -621.561,Z 491.250,A 0.000,B 0.000,C 90.000,E1 80.971} C_DIS
LIN {X -0.029,Y -615.881,Z 491.246,A 0.000,B 0.000,C 90.000,E1 80.330} C_DIS
LIN {X -0.052,Y -609.748,Z 491.243,A 0.000,B 0.000,C 90.000,E1 79.690} C_DIS
LIN {X 0.179,Y -605.903,Z 491.241,A 0.000,B 0.000,C 90.000,E1 79.285} C_DIS
LIN {X -0.256,Y -598.221,Z 491.237,A 0.000,B 0.000,C 90.000,E1 78.634} C_DIS
LIN {X 0.284,Y -594.085,Z 491.235,A 0.000,B 0.000,C 90.000,E1 78.229} C_DIS
LIN {X -0.019,Y -588.089,Z 491.232,A 0.000,B 0.000,C 90.000,E1 77.813} C_DIS
LIN {X 0.313,Y -583.511,Z 491.231,A 0.000,B 0.000,C 90.000,E1 77.465} C_DIS
LIN {X 0.130,Y -577.554,Z 491.229,A 0.000,B 0.000,C 90.000,E1 77.117} C_DIS
LIN {X 0.185,Y -572.378,Z 491.227,A 0.000,B 0.000,C 90.000,E1 76.825} C_DIS
LIN {X 0.016,Y -566.901,Z 491.226,A 0.000,B 0.000,C 90.000,E1 76.589} C_DIS
LIN {X 0.089,Y -559.951,Z 491.224,A 0.000,B 0.000,C 90.000,E1 76.297} C_DIS
LIN {X 0.051,Y -552.465,Z 491.223,A 0.000,B 0.000,C 90.000,E1 76.061} C_DIS
LIN {X -0.266,Y -545.989,Z 491.222,A 0.000,B 0.000,C 90.000,E1 75.936} C_DIS
LIN {X -0.149,Y -539.446,Z 491.221,A 0.000,B 0.000,C 90.000,E1 75.811} C_DIS
LIN {X -0.172,Y -534.597,Z 491.221,A 0.000,B 0.000,C 90.000,E1 75.755} C_DIS
LIN {X -0.016,Y -522.153,Z 491.220,A 0.000,B 0.000,C 90.000,E1 75.644} C_DIS
LIN {X -0.087,Y -519.387,Z 491.220,A 0.000,B 0.000,C 90.000,E1 75.644} C_DIS
LIN {X -0.113,Y -478.574,Z 491.220,A 0.000,B 0.000,C 90.000,E1 75.644} C_DIS
LIN {X 0.231,Y -474.160,Z 491.201,A 0.000,B 0.000,C 90.000,E1 72.054} C_DIS
LIN {X 0.097,Y -465.645,Z 491.173,A 0.000,B 0.000,C 90.000,E1 67.050} C_DIS
LIN {X -0.024,Y -456.639,Z 491.148,A 0.000,B 0.000,C 90.000,E1 62.615} C_DIS
LIN {X -0.024,Y -455.595,Z 491.144,A 0.000,B 0.000,C 90.000,E1 61.975} C_DIS
LIN {X 0.063,Y -453.279,Z 491.139,A 0.000,B 0.000,C 90.000,E1 61.001} C_DIS
LIN {X 0.094,Y -451.703,Z 491.135,A 0.000,B 0.000,C 90.000,E1 60.333} C_DIS
LIN {X 0.055,Y -451.722,Z 491.135,A 0.000,B 0.000,C 90.000,E1 60.333} C_DIS
LIN {X -0.110,Y -457.476,Z 491.129,A 0.000,B 0.000,C 90.000,E1 59.253} C_DIS
LIN {X -0.137,Y -461.384,Z 491.125,A 0.000,B 0.000,C 90.000,E1 58.456} C_DIS
LIN {X 0.122,Y -464.275,Z 491.121,A 0.000,B 0.000,C 90.000,E1 57.788} C_DIS
LIN {X 0.012,Y -466.944,Z 491.118,A 0.000,B 0.000,C 90.000,E1 57.168} C_DIS
LIN {X -0.077,Y -469.389,Z 491.114,A 0.000,B 0.000,C 90.000,E1 56.548} C_DIS
LIN {X -0.150,Y -471.498,Z 491.111,A 0.000,B 0.000,C 90.000,E1 55.928} C_DIS
LIN {X -0.041,Y -474.197,Z 491.105,A 0.000,B 0.000,C 90.000,E1 54.975} C_DIS
LIN {X -0.083,Y -475.696,Z 491.102,A 0.000,B 0.000,C 90.000,E1 54.356} C_DIS
LIN {X -0.041,Y -477.512,Z 491.097,A 0.000,B 0.000,C 90.000,E1 53.417} C_DIS
LIN {X 0.028,Y -478.942,Z 491.092,A 0.000,B 0.000,C 90.000,E1 52.477} C_DIS
LIN {X 0.011,Y -479.780,Z 491.088,A 0.000,B 0.000,C 90.000,E1 51.859} C_DIS
LIN {X 0.027,Y -480.762,Z 491.083,A 0.000,B 0.000,C 90.000,E1 50.928} C_DIS
LIN {X -0.062,Y -481.717,Z 491.076,A 0.000,B 0.000,C 90.000,E1 49.703} C_DIS
LIN {X -0.134,Y -482.209,Z 491.073,A 0.000,B 0.000,C 90.000,E1 49.094} C_DIS
LIN {X 0.058,Y -482.828,Z 491.066,A 0.000,B 0.000,C 90.000,E1 47.838} C_DIS
LIN {X -0.004,Y -483.128,Z 491.062,A 0.000,B 0.000,C 90.000,E1 47.229} C_DIS
LIN {X 0.206,Y -483.369,Z 491.056,A 0.000,B 0.000,C 90.000,E1 45.972} C_DIS
LIN {X 0.071,Y -483.435,Z 491.049,A 0.000,B 0.000,C 90.000,E1 44.757} C_DIS
LIN {X 0.071,Y -483.281,Z 491.040,A 0.000,B 0.000,C 90.000,E1 43.218} C_DIS
LIN {X -0.048,Y -482.830,Z 491.033,A 0.000,B 0.000,C 90.000,E1 42.000} C_DIS
LIN {X 0.022,Y -482.389,Z 491.028,A 0.000,B 0.000,C 90.000,E1 41.067} C_DIS
LIN {X 0.191,Y -481.311,Z 491.018,A 0.000,B 0.000,C 90.000,E1 39.197} C_DIS
LIN {X 0.029,Y -480.231,Z 491.008,A 0.000,B 0.000,C 90.000,E1 37.363} C_DIS
LIN {X -0.069,Y -479.442,Z 491.001,A 0.000,B 0.000,C 90.000,E1 36.137} C_DIS
LIN {X -0.072,Y -477.924,Z 490.990,A 0.000,B 0.000,C 90.000,E1 34.278} C_DIS
LIN {X 0.110,Y -476.571,Z 490.982,A 0.000,B 0.000,C 90.000,E1 32.704} C_DIS
LIN {X 0.038,Y -474.771,Z 490.971,A 0.000,B 0.000,C 90.000,E1 30.846} C_DIS
LIN {X 0.245,Y -472.835,Z 490.961,A 0.000,B 0.000,C 90.000,E1 28.949} C_DIS
LIN {X -0.226,Y -470.933,Z 490.951,A 0.000,B 0.000,C 90.000,E1 27.129} C_DIS
LIN {X 0.094,Y -469.228,Z 490.940,A 0.000,B 0.000,C 90.000,E1 25.207} C_DIS
LIN {X -0.057,Y -466.741,Z 490.923,A 0.000,B 0.000,C 90.000,E1 22.078} C_DIS
LIN {X 0.025,Y -465.626,Z 490.912,A 0.000,B 0.000,C 90.000,E1 20.174} C_DIS
LIN {X 0.146,Y -464.497,Z 490.900,A 0.000,B 0.000,C 90.000,E1 17.946} C_DIS
LIN {X -0.126,Y -463.589,Z 490.889,A 0.000,B 0.000,C 90.000,E1 16.079} C_DIS
LIN {X -0.176,Y -462.574,Z 490.873,A 0.000,B 0.000,C 90.000,E1 13.231} C_DIS
LIN {X 0.120,Y -462.058,Z 490.856,A 0.000,B 0.000,C 90.000,E1 10.018} C_DIS
LIN {X 0.142,Y -462.187,Z 490.842,A 0.000,B 0.000,C 90.000,E1 7.473} C_DIS
LIN {X -0.114,Y -463.244,Z 490.822,A 0.000,B 0.000,C 90.000,E1 4.012} C_DIS
LIN {X -0.219,Y -464.646,Z 490.808,A 0.000,B 0.000,C 90.000,E1 1.489} C_DIS
LIN {X -0.076,Y -466.771,Z 490.794,A 0.000,B 0.000,C 90.000,E1 358.854} C_DIS
LIN {X 0.175,Y -469.639,Z 490.778,A 0.000,B 0.000,C 90.000,E1 355.988} C_DIS
LIN {X -0.173,Y -471.920,Z 490.767,A 0.000,B 0.000,C 90.000,E1 354.147} C_DIS
LIN {X 0.053,Y -474.382,Z 490.757,A 0.000,B 0.000,C 90.000,E1 352.243} C_DIS
LIN {X -0.064,Y -478.312,Z 490.741,A 0.000,B 0.000,C 90.000,E1 349.454} C_DIS
LIN {X -0.019,Y -484.108,Z 490.723,A 0.000,B 0.000,C 90.000,E1 346.047} C_DIS
LIN {X -0.084,Y -487.850,Z 490.712,A 0.000,B 0.000,C 90.000,E1 344.212} C_DIS
LIN {X 0.091,Y -492.414,Z 490.700,A 0.000,B 0.000,C 90.000,E1 342.054} C_DIS
LIN {X 0.021,Y -496.439,Z 490.690,A 0.000,B 0.000,C 90.000,E1 340.242} C_DIS
LIN {X 0.136,Y -499.888,Z 490.682,A 0.000,B 0.000,C 90.000,E1 338.720} C_DIS
LIN {X 0.030,Y -503.233,Z 490.674,A 0.000,B 0.000,C 90.000,E1 337.230} C_DIS
LIN {X 0.071,Y -507.175,Z 490.664,A 0.000,B 0.000,C 90.000,E1 335.433} C_DIS
LIN {X -0.260,Y -509.691,Z 490.657,A 0.000,B 0.000,C 90.000,E1 334.280} C_DIS
LIN {X -0.111,Y -513.447,Z 490.647,A 0.000,B 0.000,C 90.000,E1 332.487} C_DIS
LIN {X -0.090,Y -517.286,Z 490.637,A 0.000,B 0.000,C 90.000,E1 330.717} C_DIS
LIN {X -0.109,Y -522.605,Z 490.624,A 0.000,B 0.000,C 90.000,E1 328.377} C_DIS
LIN {X 0.305,Y -528.042,Z 490.611,A 0.000,B 0.000,C 90.000,E1 326.008} C_DIS
LIN {X -0.135,Y -532.876,Z 490.600,A 0.000,B 0.000,C 90.000,E1 324.036} C_DIS
LIN {X 0.278,Y -536.349,Z 490.592,A 0.000,B 0.000,C 90.000,E1 322.557} C_DIS
LIN {X -0.104,Y -539.802,Z 490.584,A 0.000,B 0.000,C 90.000,E1 321.170} C_DIS
LIN {X -0.060,Y -543.906,Z 490.575,A 0.000,B 0.000,C 90.000,E1 319.461} C_DIS
LIN {X 0.027,Y -547.293,Z 490.567,A 0.000,B 0.000,C 90.000,E1 318.038} C_DIS
LIN {X -0.230,Y -551.226,Z 490.558,A 0.000,B 0.000,C 90.000,E1 316.377} C_DIS
LIN {X -0.012,Y -555.023,Z 490.548,A 0.000,B 0.000,C 90.000,E1 314.676} C_DIS
LIN {X 0.355,Y -559.379,Z 490.537,A 0.000,B 0.000,C 90.000,E1 312.690} C_DIS
LIN {X -0.021,Y -563.148,Z 490.528,A 0.000,B 0.000,C 90.000,E1 311.067} C_DIS
LIN {X 0.099,Y -566.805,Z 490.519,A 0.000,B 0.000,C 90.000,E1 309.402} C_DIS
LIN {X 0.377,Y -570.441,Z 490.510,A 0.000,B 0.000,C 90.000,E1 307.729} C_DIS
LIN {X -0.070,Y -574.186,Z 490.501,A 0.000,B 0.000,C 90.000,E1 306.137} C_DIS
LIN {X 0.157,Y -578.036,Z 490.492,A 0.000,B 0.000,C 90.000,E1 304.485} C_DIS
LIN {X -0.170,Y -581.249,Z 490.484,A 0.000,B 0.000,C 90.000,E1 303.166} C_DIS
LIN {X -0.100,Y -584.983,Z 490.475,A 0.000,B 0.000,C 90.000,E1 301.544} C_DIS
LIN {X 0.042,Y -588.310,Z 490.466,A 0.000,B 0.000,C 90.000,E1 299.922} C_DIS
LIN {X -0.236,Y -590.871,Z 490.459,A 0.000,B 0.000,C 90.000,E1 298.615} C_DIS
LIN {X 0.152,Y -592.745,Z 490.453,A 0.000,B 0.000,C 90.000,E1 297.513} C_DIS
LIN {X -0.325,Y -594.772,Z 490.446,A 0.000,B 0.000,C 90.000,E1 296.232} C_DIS
LIN {X -0.147,Y -596.131,Z 490.440,A 0.000,B 0.000,C 90.000,E1 295.155} C_DIS
LIN {X 0.051,Y -597.254,Z 490.434,A 0.000,B 0.000,C 90.000,E1 294.079} C_DIS
LIN {X -0.062,Y -598.417,Z 490.427,A 0.000,B 0.000,C 90.000,E1 292.770} C_DIS
LIN {X -0.160,Y -599.475,Z 490.419,A 0.000,B 0.000,C 90.000,E1 291.461} C_DIS
LIN {X 0.096,Y -600.401,Z 490.412,A 0.000,B 0.000,C 90.000,E1 290.120} C_DIS
LIN {X -0.198,Y -601.081,Z 490.405,A 0.000,B 0.000,C 90.000,E1 288.833} C_DIS
LIN {X -0.099,Y -601.994,Z 490.394,A 0.000,B 0.000,C 90.000,E1 286.985} C_DIS
LIN {X -0.268,Y -602.629,Z 490.386,A 0.000,B 0.000,C 90.000,E1 285.426} C_DIS
LIN {X -0.047,Y -603.018,Z 490.380,A 0.000,B 0.000,C 90.000,E1 284.356} C_DIS
LIN {X -0.239,Y -603.323,Z 490.372,A 0.000,B 0.000,C 90.000,E1 283.063} C_DIS
LIN {X -0.152,Y -603.537,Z 490.367,A 0.000,B 0.000,C 90.000,E1 282.007} C_DIS
LIN {X 0.252,Y -603.660,Z 490.359,A 0.000,B 0.000,C 90.000,E1 280.658} C_DIS
LIN {X -0.054,Y -603.581,Z 490.352,A 0.000,B 0.000,C 90.000,E1 279.378} C_DIS
LIN {X 0.140,Y -603.352,Z 490.345,A 0.000,B 0.000,C 90.000,E1 278.049} C_DIS
LIN {X 0.103,Y -603.001,Z 490.339,A 0.000,B 0.000,C 90.000,E1 277.004} C_DIS
LIN {X -0.019,Y -602.509,Z 490.333,A 0.000,B 0.000,C 90.000,E1 275.967} C_DIS
LIN {X -0.202,Y -601.848,Z 490.327,A 0.000,B 0.000,C 90.000,E1 274.935} C_DIS
LIN {X 0.259,Y -601.047,Z 490.322,A 0.000,B 0.000,C 90.000,E1 273.841} C_DIS
LIN {X -0.295,Y -599.810,Z 490.314,A 0.000,B 0.000,C 90.000,E1 272.579} C_DIS
LIN {X -0.272,Y -598.206,Z 490.307,A 0.000,B 0.000,C 90.000,E1 271.260} C_DIS
LIN {X -0.290,Y -596.437,Z 490.300,A 0.000,B 0.000,C 90.000,E1 269.943} C_DIS
LIN {X 0.256,Y -594.502,Z 490.292,A 0.000,B 0.000,C 90.000,E1 268.568} C_DIS
LIN {X -0.196,Y -592.011,Z 490.283,A 0.000,B 0.000,C 90.000,E1 267.020} C_DIS
LIN {X -0.272,Y -589.827,Z 490.276,A 0.000,B 0.000,C 90.000,E1 265.698} C_DIS
LIN {X 0.206,Y -587.378,Z 490.269,A 0.000,B 0.000,C 90.000,E1 264.318} C_DIS
LIN {X 0.047,Y -584.770,Z 490.261,A 0.000,B 0.000,C 90.000,E1 262.996} C_DIS
LIN {X -0.009,Y -582.179,Z 490.254,A 0.000,B 0.000,C 90.000,E1 261.659} C_DIS
LIN {X 0.033,Y -579.090,Z 490.245,A 0.000,B 0.000,C 90.000,E1 260.038} C_DIS
LIN {X -0.219,Y -576.864,Z 490.239,A 0.000,B 0.000,C 90.000,E1 258.982} C_DIS
LIN {X -0.201,Y -573.329,Z 490.230,A 0.000,B 0.000,C 90.000,E1 257.353} C_DIS
LIN {X -0.205,Y -570.338,Z 490.222,A 0.000,B 0.000,C 90.000,E1 255.992} C_DIS
LIN {X -0.255,Y -567.170,Z 490.215,A 0.000,B 0.000,C 90.000,E1 254.629} C_DIS
LIN {X 0.018,Y -564.531,Z 490.208,A 0.000,B 0.000,C 90.000,E1 253.504} C_DIS
LIN {X -0.129,Y -561.783,Z 490.202,A 0.000,B 0.000,C 90.000,E1 252.417} C_DIS
LIN {X -0.184,Y -558.226,Z 490.195,A 0.000,B 0.000,C 90.000,E1 251.040} C_DIS
LIN {X -0.230,Y -555.164,Z 490.188,A 0.000,B 0.000,C 90.000,E1 249.934} C_DIS
LIN {X -0.231,Y -551.176,Z 490.181,A 0.000,B 0.000,C 90.000,E1 248.539} C_DIS
LIN {X 0.074,Y -548.701,Z 490.176,A 0.000,B 0.000,C 90.000,E1 247.667} C_DIS
LIN {X -0.140,Y -544.408,Z 490.168,A 0.000,B 0.000,C 90.000,E1 246.282} C_DIS
LIN {X -0.162,Y -540.828,Z 490.162,A 0.000,B 0.000,C 90.000,E1 245.153} C_DIS
LIN {X -0.031,Y -536.252,Z 490.154,A 0.000,B 0.000,C 90.000,E1 243.717} C_DIS
LIN {X 0.008,Y -531.585,Z 490.146,A 0.000,B 0.000,C 90.000,E1 242.281} C_DIS
LIN {X 0.126,Y -525.974,Z 490.136,A 0.000,B 0.000,C 90.000,E1 240.539} C_DIS
LIN {X 0.239,Y -521.347,Z 490.128,A 0.000,B 0.000,C 90.000,E1 239.076} C_DIS
LIN {X 0.191,Y -515.740,Z 490.119,A 0.000,B 0.000,C 90.000,E1 237.327} C_DIS
LIN {X -0.310,Y -512.802,Z 490.114,A 0.000,B 0.000,C 90.000,E1 236.501} C_DIS
LIN {X -0.077,Y -505.829,Z 490.102,A 0.000,B 0.000,C 90.000,E1 234.402} C_DIS
LIN {X 0.011,Y -497.077,Z 490.087,A 0.000,B 0.000,C 90.000,E1 231.698} C_DIS
LIN {X -0.055,Y -492.616,Z 490.079,A 0.000,B 0.000,C 90.000,E1 230.194} C_DIS
LIN {X -0.194,Y -488.238,Z 490.070,A 0.000,B 0.000,C 90.000,E1 228.690} C_DIS
LIN {X -0.146,Y -482.287,Z 490.059,A 0.000,B 0.000,C 90.000,E1 226.539} C_DIS
LIN {X 0.054,Y -476.507,Z 490.046,A 0.000,B 0.000,C 90.000,E1 224.352} C_DIS
LIN {X 0.028,Y -471.812,Z 490.036,A 0.000,B 0.000,C 90.000,E1 222.486} C_DIS
LIN {X -0.104,Y -467.297,Z 490.026,A 0.000,B 0.000,C 90.000,E1 220.620} C_DIS
LIN {X -0.051,Y -463.722,Z 490.017,A 0.000,B 0.000,C 90.000,E1 219.036} C_DIS
LIN {X 0.130,Y -459.001,Z 490.005,A 0.000,B 0.000,C 90.000,E1 216.790} C_DIS
LIN {X -0.080,Y -455.101,Z 489.994,A 0.000,B 0.000,C 90.000,E1 214.898} C_DIS
LIN {X -0.002,Y -451.319,Z 489.983,A 0.000,B 0.000,C 90.000,E1 212.959} C_DIS
LIN {X 0.120,Y -447.741,Z 489.972,A 0.000,B 0.000,C 90.000,E1 211.003} C_DIS
LIN {X -0.073,Y -444.177,Z 489.962,A 0.000,B 0.000,C 90.000,E1 209.077} C_DIS
LIN {X -0.138,Y -440.086,Z 489.949,A 0.000,B 0.000,C 90.000,E1 206.796} C_DIS
LIN {X -0.170,Y -437.101,Z 489.940,A 0.000,B 0.000,C 90.000,E1 205.155} C_DIS
LIN {X -0.028,Y -433.564,Z 489.929,A 0.000,B 0.000,C 90.000,E1 203.153} C_DIS
LIN {X 0.232,Y -429.543,Z 489.916,A 0.000,B 0.000,C 90.000,E1 200.791} C_DIS
LIN {X -0.074,Y -425.889,Z 489.903,A 0.000,B 0.000,C 90.000,E1 198.489} C_DIS
LIN {X 0.145,Y -422.892,Z 489.892,A 0.000,B 0.000,C 90.000,E1 196.441} C_DIS
LIN {X -0.008,Y -420.637,Z 489.882,A 0.000,B 0.000,C 90.000,E1 194.773} C_DIS
LIN {X -0.047,Y -417.281,Z 489.867,A 0.000,B 0.000,C 90.000,E1 192.063} C_DIS
LIN {X -0.055,Y -414.901,Z 489.856,A 0.000,B 0.000,C 90.000,E1 190.018} C_DIS
LIN {X -0.180,Y -411.968,Z 489.840,A 0.000,B 0.000,C 90.000,E1 187.296} C_DIS
LIN {X -0.094,Y -409.996,Z 489.829,A 0.000,B 0.000,C 90.000,E1 185.220} C_DIS
LIN {X -0.134,Y -407.513,Z 489.814,A 0.000,B 0.000,C 90.000,E1 182.465} C_DIS
LIN {X 0.126,Y -405.562,Z 489.798,A 0.000,B 0.000,C 90.000,E1 179.656} C_DIS
LIN {X -0.083,Y -404.147,Z 489.783,A 0.000,B 0.000,C 90.000,E1 176.906} C_DIS
LIN {X 0.074,Y -403.203,Z 489.762,A 0.000,B 0.000,C 90.000,E1 173.053} C_DIS
LIN {X 0.073,Y -403.335,Z 489.742,A 0.000,B 0.000,C 90.000,E1 169.567} C_DIS
LIN {X -0.156,Y -404.180,Z 489.725,A 0.000,B 0.000,C 90.000,E1 166.464} C_DIS
LIN {X -0.179,Y -405.378,Z 489.709,A 0.000,B 0.000,C 90.000,E1 163.685} C_DIS
LIN {X -0.099,Y -407.285,Z 489.692,A 0.000,B 0.000,C 90.000,E1 160.550} C_DIS
LIN {X 0.085,Y -409.144,Z 489.678,A 0.000,B 0.000,C 90.000,E1 158.103} C_DIS
LIN {X -0.028,Y -411.037,Z 489.667,A 0.000,B 0.000,C 90.000,E1 156.049} C_DIS
LIN {X -0.008,Y -413.370,Z 489.654,A 0.000,B 0.000,C 90.000,E1 153.640} C_DIS
LIN {X 0.207,Y -415.126,Z 489.644,A 0.000,B 0.000,C 90.000,E1 151.897} C_DIS
LIN {X 0.087,Y -416.767,Z 489.635,A 0.000,B 0.000,C 90.000,E1 150.205} C_DIS
LIN {X -0.248,Y -419.043,Z 489.621,A 0.000,B 0.000,C 90.000,E1 147.867} C_DIS
LIN {X 0.004,Y -420.595,Z 489.612,A 0.000,B 0.000,C 90.000,E1 146.135} C_DIS
LIN {X -0.088,Y -422.465,Z 489.601,A 0.000,B 0.000,C 90.000,E1 144.116} C_DIS
LIN {X -0.011,Y -424.691,Z 489.587,A 0.000,B 0.000,C 90.000,E1 141.743} C_DIS
LIN {X -0.035,Y -425.928,Z 489.580,A 0.000,B 0.000,C 90.000,E1 140.400} C_DIS
LIN {X 0.054,Y -426.867,Z 489.574,A 0.000,B 0.000,C 90.000,E1 139.380} C_DIS
LIN {X 0.055,Y -427.939,Z 489.567,A 0.000,B 0.000,C 90.000,E1 138.038} C_DIS
LIN {X 0.037,Y -428.843,Z 489.560,A 0.000,B 0.000,C 90.000,E1 136.701} C_DIS
LIN {X 0.032,Y -429.595,Z 489.552,A 0.000,B 0.000,C 90.000,E1 135.364} C_DIS
LIN {X 0.038,Y -430.042,Z 489.545,A 0.000,B 0.000,C 90.000,E1 134.028} C_DIS
LIN {X 0.130,Y -430.243,Z 489.539,A 0.000,B 0.000,C 90.000,E1 133.014} C_DIS
LIN {X 0.150,Y -430.002,Z 489.532,A 0.000,B 0.000,C 90.000,E1 131.676} C_DIS
LIN {X -0.044,Y -429.528,Z 489.526,A 0.000,B 0.000,C 90.000,E1 130.701} C_DIS
LIN {X 0.004,Y -428.444,Z 489.519,A 0.000,B 0.000,C 90.000,E1 129.358} C_DIS
LIN {X 0.028,Y -427.054,Z 489.511,A 0.000,B 0.000,C 90.000,E1 128.016} C_DIS
LIN {X 0.103,Y -425.432,Z 489.504,A 0.000,B 0.000,C 90.000,E1 126.664} C_DIS
LIN {X -0.220,Y -423.072,Z 489.494,A 0.000,B 0.000,C 90.000,E1 125.025} C_DIS
LIN {X 0.053,Y -421.107,Z 489.487,A 0.000,B 0.000,C 90.000,E1 123.658} C_DIS
LIN {X 0.015,Y -421.111,Z 489.487,A 0.000,B 0.000,C 90.000,E1 123.658} C_DIS
LIN {X 0.154,Y -430.791,Z 489.468,A 0.000,B 0.000,C 90.000,E1 120.256} C_DIS
LIN {X 0.114,Y -440.753,Z 489.446,A 0.000,B 0.000,C 90.000,E1 116.283} C_DIS
LIN {X 0.084,Y -444.618,Z 489.439,A 0.000,B 0.000,C 90.000,E1 114.975} C_DIS
LIN {X 0.140,Y -455.476,Z 489.414,A 0.000,B 0.000,C 90.000,E1 110.429} C_DIS
LIN {X -0.062,Y -457.264,Z 489.410,A 0.000,B 0.000,C 90.000,E1 109.812} C_DIS
LIN {X 0.006,Y -465.885,Z 489.387,A 0.000,B 0.000,C 90.000,E1 105.662} C_DIS
LIN {X -0.223,Y -467.708,Z 489.383,A 0.000,B 0.000,C 90.000,E1 104.954} C_DIS
LIN {X -0.251,Y -467.777,Z 489.383,A 0.000,B 0.000,C 90.000,E1 104.954} C_DIS
LIN {X -0.118,Y -477.694,Z 489.382,A 0.000,B 0.000,C 90.000,E1 104.828} C_DIS
LIN {X -0.018,Y -485.427,Z 489.382,A 0.000,B 0.000,C 90.000,E1 104.717} C_DIS
LIN {X -0.024,Y -503.801,Z 489.380,A 0.000,B 0.000,C 90.000,E1 104.411} C_DIS
LIN {X -0.241,Y -510.406,Z 489.379,A 0.000,B 0.000,C 90.000,E1 104.300} C_DIS
LIN {X -0.105,Y -524.138,Z 489.377,A 0.000,B 0.000,C 90.000,E1 103.939} C_DIS
LIN {X -0.027,Y -534.724,Z 489.376,A 0.000,B 0.000,C 90.000,E1 103.647} C_DIS
LIN {X -0.245,Y -545.138,Z 489.374,A 0.000,B 0.000,C 90.000,E1 103.355} C_DIS
LIN {X -0.233,Y -554.630,Z 489.372,A 0.000,B 0.000,C 90.000,E1 103.008} C_DIS
LIN {X 0.014,Y -561.125,Z 489.371,A 0.000,B 0.000,C 90.000,E1 102.715} C_DIS
LIN {X 0.137,Y -567.712,Z 489.369,A 0.000,B 0.000,C 90.000,E1 102.411} C_DIS
LIN {X -0.078,Y -574.056,Z 489.367,A 0.000,B 0.000,C 90.000,E1 102.119} C_DIS
LIN {X -0.049,Y -577.122,Z 489.366,A 0.000,B 0.000,C 90.000,E1 101.951} C_DIS
LIN {X -0.210,Y -586.427,Z 489.363,A 0.000,B 0.000,C 90.000,E1 101.422} C_DIS
LIN {X -0.205,Y -590.509,Z 489.362,A 0.000,B 0.000,C 90.000,E1 101.130} C_DIS
LIN {X -0.013,Y -592.201,Z 489.361,A 0.000,B 0.000,C 90.000,E1 101.007} C_DIS
LIN {X -0.006,Y -597.958,Z 489.359,A 0.000,B 0.000,C 90.000,E1 100.602} C_DIS
LIN {X -0.106,Y -605.397,Z 489.356,A 0.000,B 0.000,C 90.000,E1 100.018} C_DIS
LIN {X 0.224,Y -610.371,Z 489.353,A 0.000,B 0.000,C 90.000,E1 99.557} C_DIS
LIN {X 0.093,Y -616.659,Z 489.350,A 0.000,B 0.000,C 90.000,E1 98.973} C_DIS
LIN {X 0.127,Y -622.595,Z 489.346,A 0.000,B 0.000,C 90.000,E1 98.341} C_DIS
LIN {X 0.136,Y -627.885,Z 489.343,A 0.000,B 0.000,C 90.000,E1 97.701} C_DIS
LIN {X 0.103,Y -632.637,Z 489.339,A 0.000,B 0.000,C 90.000,E1 97.068} C_DIS
LIN {X 0.052,Y -637.637,Z 489.335,A 0.000,B 0.000,C 90.000,E1 96.315} C_DIS
LIN {X 0.104,Y -641.331,Z 489.332,A 0.000,B 0.000,C 90.000,E1 95.682} C_DIS
LIN {X 0.188,Y -644.709,Z 489.328,A 0.000,B 0.000,C 90.000,E1 95.049} C_DIS
LIN {X 0.188,Y -648.396,Z 489.324,A 0.000,B 0.000,C 90.000,E1 94.302} C_DIS
LIN {X -0.213,Y -650.625,Z 489.321,A 0.000,B 0.000,C 90.000,E1 93.841} C_DIS
LIN {X 0.006,Y -652.606,Z 489.319,A 0.000,B 0.000,C 90.000,E1 93.326} C_DIS
LIN {X 0.277,Y -654.373,Z 489.316,A 0.000,B 0.000,C 90.000,E1 92.808} C_DIS
LIN {X -0.126,Y -655.845,Z 489.313,A 0.000,B 0.000,C 90.000,E1 92.350} C_DIS
LIN {X 0.139,Y -657.033,Z 489.310,A 0.000,B 0.000,C 90.000,E1 91.835} C_DIS
LIN {X -0.226,Y -657.967,Z 489.308,A 0.000,B 0.000,C 90.000,E1 91.375} C_DIS
LIN {X 0.055,Y -658.595,Z 489.305,A 0.000,B 0.000,C 90.000,E1 90.859} C_DIS
LIN {X -0.316,Y -658.980,Z 489.302,A 0.000,B 0.000,C 90.000,E1 90.401} C_DIS
LIN {X 0.159,Y -659.147,Z 489.301,A 0.000,B 0.000,C 90.000,E1 90.115} C_DIS
LIN {X 0.267,Y -659.059,Z 489.297,A 0.000,B 0.000,C 90.000,E1 89.370} C_DIS
LIN {X -0.286,Y -658.412,Z 489.293,A 0.000,B 0.000,C 90.000,E1 88.682} C_DIS
LIN {X 0.186,Y -658.173,Z 489.291,A 0.000,B 0.000,C 90.000,E1 88.396} C_DIS
LIN {X -0.167,Y -657.315,Z 489.289,A 0.000,B 0.000,C 90.000,E1 87.936} C_DIS
LIN {X -0.084,Y -655.648,Z 489.284,A 0.000,B 0.000,C 90.000,E1 87.192} C_DIS
LIN {X 0.213,Y -654.183,Z 489.282,A 0.000,B 0.000,C 90.000,E1 86.674} C_DIS
LIN {X -0.190,Y -652.455,Z 489.279,A 0.000,B 0.000,C 90.000,E1 86.216} C_DIS
LIN {X -0.123,Y -649.454,Z 489.275,A 0.000,B 0.000,C 90.000,E1 85.469} C_DIS
LIN {X 0.026,Y -646.555,Z 489.271,A 0.000,B 0.000,C 90.000,E1 84.837} C_DIS
LIN {X 0.147,Y -643.228,Z 489.268,A 0.000,B 0.000,C 90.000,E1 84.204} C_DIS
LIN {X 0.236,Y -639.492,Z 489.264,A 0.000,B 0.000,C 90.000,E1 83.571} C_DIS
LIN {X -0.208,Y -636.262,Z 489.262,A 0.000,B 0.000,C 90.000,E1 83.109} C_DIS
LIN {X -0.097,Y -631.704,Z 489.258,A 0.000,B 0.000,C 90.000,E1 82.470} C_DIS
LIN {X -0.108,Y -626.798,Z 489.255,A 0.000,B 0.000,C 90.000,E1 81.837} C_DIS
LIN {X -0.048,Y -621.567,Z 489.251,A 0.000,B 0.000,C 90.000,E1 81.197} C_DIS
LIN {X -0.054,Y -615.750,Z 489.248,A 0.000,B 0.000,C 90.000,E1 80.557} C_DIS
LIN {X 0.073,Y -610.804,Z 489.245,A 0.000,B 0.000,C 90.000,E1 80.038} C_DIS
LIN {X 0.283,Y -604.335,Z 489.241,A 0.000,B 0.000,C 90.000,E1 79.398} C_DIS
LIN {X 0.114,Y -598.969,Z 489.239,A 0.000,B 0.000,C 90.000,E1 78.926} C_DIS
LIN {X 0.026,Y -594.747,Z 489.237,A 0.000,B 0.000,C 90.000,E1 78.578} C_DIS
LIN {X 0.156,Y -588.709,Z 489.234,A 0.000,B 0.000,C 90.000,E1 78.117} C_DIS
LIN {X 0.110,Y -582.569,Z 489.232,A 0.000,B 0.000,C 90.000,E1 77.701} C_DIS
LIN {X -0.172,Y -574.854,Z 489.229,A 0.000,B 0.000,C 90.000,E1 77.285} C_DIS
LIN {X 0.240,Y -571.285,Z 489.228,A 0.000,B 0.000,C 90.000,E1 77.061} C_DIS
LIN {X -0.311,Y -564.641,Z 489.227,A 0.000,B 0.000,C 90.000,E1 76.825} C_DIS
LIN {X -0.152,Y -558.876,Z 489.225,A 0.000,B 0.000,C 90.000,E1 76.589} C_DIS
LIN {X -0.081,Y -553.079,Z 489.224,A 0.000,B 0.000,C 90.000,E1 76.408} C_DIS
LIN {X 0.258,Y -546.766,Z 489.224,A 0.000,B 0.000,C 90.000,E1 76.228} C_DIS
LIN {X -0.243,Y -540.549,Z 489.223,A 0.000,B 0.000,C 90.000,E1 76.172} C_DIS
LIN {X -0.302,Y -533.838,Z 489.223,A 0.000,B 0.000,C 90.000,E1 76.117} C_DIS
LIN {X -0.078,Y -525.098,Z 489.222,A 0.000,B 0.000,C 90.000,E1 76.047} C_DIS
LIN {X 0.160,Y -515.231,Z 489.222,A 0.000,B 0.000,C 90.000,E1 75.992} C_DIS
LIN {X 0.102,Y -479.151,Z 489.222,A 0.000,B 0.000,C 90.000,E1 75.992} C_DIS
LIN {X 0.028,Y -473.954,Z 489.200,A 0.000,B 0.000,C 90.000,E1 71.945} C_DIS
LIN {X 0.154,Y -466.326,Z 489.175,A 0.000,B 0.000,C 90.000,E1 67.539} C_DIS
LIN {X 0.038,Y -465.354,Z 489.172,A 0.000,B 0.000,C 90.000,E1 66.922} C_DIS
LIN {X 0.007,Y -456.948,Z 489.149,A 0.000,B 0.000,C 90.000,E1 62.794} C_DIS
LIN {X -0.097,Y -455.338,Z 489.144,A 0.000,B 0.000,C 90.000,E1 61.847} C_DIS
LIN {X 0.002,Y -452.157,Z 489.136,A 0.000,B 0.000,C 90.000,E1 60.539} C_DIS
LIN {X -0.038,Y -452.182,Z 489.136,A 0.000,B 0.000,C 90.000,E1 60.539} C_DIS
LIN {X 0.114,Y -458.088,Z 489.130,A 0.000,B 0.000,C 90.000,E1 59.410} C_DIS
LIN {X 0.091,Y -462.119,Z 489.126,A 0.000,B 0.000,C 90.000,E1 58.614} C_DIS
LIN {X -0.042,Y -465.812,Z 489.121,A 0.000,B 0.000,C 90.000,E1 57.837} C_DIS
LIN {X 0.001,Y -468.490,Z 489.118,A 0.000,B 0.000,C 90.000,E1 57.199} C_DIS
LIN {X 0.165,Y -470.374,Z 489.115,A 0.000,B 0.000,C 90.000,E1 56.707} C_DIS
LIN {X 0.098,Y -472.502,Z 489.112,A 0.000,B 0.000,C 90.000,E1 56.087} C_DIS
LIN {X -0.173,Y -475.303,Z 489.107,A 0.000,B 0.000,C 90.000,E1 55.182} C_DIS
LIN {X 0.069,Y -476.825,Z 489.103,A 0.000,B 0.000,C 90.000,E1 54.529} C_DIS
LIN {X -0.152,Y -478.659,Z 489.098,A 0.000,B 0.000,C 90.000,E1 53.623} C_DIS
LIN {X -0.070,Y -480.134,Z 489.093,A 0.000,B 0.000,C 90.000,E1 52.683} C_DIS
LIN {X 0.031,Y -481.281,Z 489.088,A 0.000,B 0.000,C 90.000,E1 51.743} C_DIS
LIN {X 0.143,Y -482.191,Z 489.082,A 0.000,B 0.000,C 90.000,E1 50.803} C_DIS
LIN {X -0.111,Y -482.872,Z 489.077,A 0.000,B 0.000,C 90.000,E1 49.908} C_DIS
LIN {X -0.043,Y -483.476,Z 489.072,A 0.000,B 0.000,C 90.000,E1 48.976} C_DIS
LIN {X 0.076,Y -483.945,Z 489.067,A 0.000,B 0.000,C 90.000,E1 48.038} C_DIS
LIN {X -0.199,Y -484.280,Z 489.062,A 0.000,B 0.000,C 90.000,E1 47.148} C_DIS
LIN {X 0.029,Y -484.462,Z 489.055,A 0.000,B 0.000,C 90.000,E1 45.891} C_DIS
LIN {X -0.232,Y -484.514,Z 489.050,A 0.000,B 0.000,C 90.000,E1 45.000} C_DIS
LIN {X -0.210,Y -484.313,Z 489.041,A 0.000,B 0.000,C 90.000,E1 43.461} C_DIS
LIN {X -0.124,Y -484.023,Z 489.036,A 0.000,B 0.000,C 90.000,E1 42.528} C_DIS
LIN {X -0.227,Y -483.445,Z 489.029,A 0.000,B 0.000,C 90.000,E1 41.310} C_DIS
LIN {X -0.029,Y -482.344,Z 489.019,A 0.000,B 0.000,C 90.000,E1 39.439} C_DIS
LIN {X -0.160,Y -481.232,Z 489.009,A 0.000,B 0.000,C 90.000,E1 37.604} C_DIS
LIN {X 0.246,Y -480.213,Z 489.000,A 0.000,B 0.000,C 90.000,E1 36.011} C_DIS
LIN {X -0.131,Y -478.649,Z 488.990,A 0.000,B 0.000,C 90.000,E1 34.199} C_DIS
LIN {X 0.062,Y -477.250,Z 488.981,A 0.000,B 0.000,C 90.000,E1 32.625} C_DIS
LIN {X -0.026,Y -475.761,Z 488.973,A 0.000,B 0.000,C 90.000,E1 31.082} C_DIS
LIN {X 0.037,Y -473.802,Z 488.962,A 0.000,B 0.000,C 90.000,E1 29.205} C_DIS
LIN {X 0.005,Y -471.836,Z 488.952,A 0.000,B 0.000,C 90.000,E1 27.334} C_DIS
LIN {X -0.072,Y -470.073,Z 488.941,A 0.000,B 0.000,C 90.000,E1 25.463} C_DIS
LIN {X -0.186,Y -467.526,Z 488.924,A 0.000,B 0.000,C 90.000,E1 22.333} C_DIS
LIN {X -0.138,Y -466.160,Z 488.912,A 0.000,B 0.000,C 90.000,E1 20.120} C_DIS
LIN {X 0.215,Y -465.155,Z 488.901,A 0.000,B 0.000,C 90.000,E1 18.181} C_DIS
LIN {X -0.045,Y -464.247,Z 488.891,A 0.000,B 0.000,C 90.000,E1 16.315} C_DIS
LIN {X -0.074,Y -463.140,Z 488.875,A 0.000,B 0.000,C 90.000,E1 13.467} C_DIS
LIN {X -0.209,Y -462.502,Z 488.857,A 0.000,B 0.000,C 90.000,E1 10.310} C_DIS
LIN {X -0.110,Y -462.539,Z 488.843,A 0.000,B 0.000,C 90.000,E1 7.757} C_DIS
LIN {X 0.062,Y -463.453,Z 488.824,A 0.000,B 0.000,C 90.000,E1 4.245} C_DIS
LIN {X 0.223,Y -464.568,Z 488.811,A 0.000,B 0.000,C 90.000,E1 2.007} C_DIS
LIN {X -0.073,Y -467.059,Z 488.794,A 0.000,B 0.000,C 90.000,E1 358.854} C_DIS
LIN {X 0.188,Y -469.900,Z 488.778,A 0.000,B 0.000,C 90.000,E1 355.988} C_DIS
LIN {X -0.154,Y -472.173,Z 488.767,A 0.000,B 0.000,C 90.000,E1 354.147} C_DIS
LIN {X -0.091,Y -475.071,Z 488.755,A 0.000,B 0.000,C 90.000,E1 351.951} C_DIS
LIN {X -0.180,Y -479.065,Z 488.740,A 0.000,B 0.000,C 90.000,E1 349.162} C_DIS
LIN {X 0.100,Y -486.275,Z 488.717,A 0.000,B 0.000,C 90.000,E1 345.117} C_DIS
LIN {X 0.220,Y -490.751,Z 488.706,A 0.000,B 0.000,C 90.000,E1 342.960} C_DIS
LIN {X 0.113,Y -494.778,Z 488.695,A 0.000,B 0.000,C 90.000,E1 341.148} C_DIS
LIN {X 0.150,Y -499.577,Z 488.684,A 0.000,B 0.000,C 90.000,E1 339.028} C_DIS
LIN {X 0.037,Y -502.984,Z 488.675,A 0.000,B 0.000,C 90.000,E1 337.539} C_DIS
LIN {X -0.294,Y -507.603,Z 488.664,A 0.000,B 0.000,C 90.000,E1 335.485} C_DIS
LIN {X -0.059,Y -510.786,Z 488.655,A 0.000,B 0.000,C 90.000,E1 333.973} C_DIS
LIN {X 0.109,Y -514.593,Z 488.646,A 0.000,B 0.000,C 90.000,E1 332.180} C_DIS
LIN {X 0.148,Y -518.450,Z 488.636,A 0.000,B 0.000,C 90.000,E1 330.411} C_DIS
LIN {X -0.240,Y -523.180,Z 488.624,A 0.000,B 0.000,C 90.000,E1 328.408} C_DIS
LIN {X 0.053,Y -525.222,Z 488.620,A 0.000,B 0.000,C 90.000,E1 327.502} C_DIS
LIN {X 0.144,Y -529.366,Z 488.610,A 0.000,B 0.000,C 90.000,E1 325.754} C_DIS
LIN {X 0.046,Y -533.550,Z 488.600,A 0.000,B 0.000,C 90.000,E1 324.036} C_DIS
LIN {X 0.047,Y -537.041,Z 488.592,A 0.000,B 0.000,C 90.000,E1 322.603} C_DIS
LIN {X 0.106,Y -540.541,Z 488.584,A 0.000,B 0.000,C 90.000,E1 321.170} C_DIS
LIN {X 0.168,Y -544.684,Z 488.575,A 0.000,B 0.000,C 90.000,E1 319.461} C_DIS
LIN {X -0.137,Y -548.108,Z 488.567,A 0.000,B 0.000,C 90.000,E1 318.081} C_DIS
LIN {X 0.032,Y -552.080,Z 488.558,A 0.000,B 0.000,C 90.000,E1 316.377} C_DIS
LIN {X 0.271,Y -555.909,Z 488.548,A 0.000,B 0.000,C 90.000,E1 314.676} C_DIS
LIN {X -0.128,Y -560.338,Z 488.538,A 0.000,B 0.000,C 90.000,E1 312.771} C_DIS
LIN {X 0.310,Y -564.129,Z 488.528,A 0.000,B 0.000,C 90.000,E1 311.067} C_DIS
LIN {X -0.022,Y -567.179,Z 488.521,A 0.000,B 0.000,C 90.000,E1 309.725} C_DIS
LIN {X 0.143,Y -570.292,Z 488.513,A 0.000,B 0.000,C 90.000,E1 308.338} C_DIS
LIN {X 0.047,Y -574.040,Z 488.504,A 0.000,B 0.000,C 90.000,E1 306.710} C_DIS
LIN {X -0.048,Y -578.523,Z 488.493,A 0.000,B 0.000,C 90.000,E1 304.818} C_DIS
LIN {X 0.282,Y -582.397,Z 488.484,A 0.000,B 0.000,C 90.000,E1 303.166} C_DIS
LIN {X -0.293,Y -585.561,Z 488.477,A 0.000,B 0.000,C 90.000,E1 301.878} C_DIS
LIN {X -0.196,Y -587.843,Z 488.471,A 0.000,B 0.000,C 90.000,E1 300.797} C_DIS
LIN {X -0.076,Y -590.047,Z 488.465,A 0.000,B 0.000,C 90.000,E1 299.716} C_DIS
LIN {X 0.193,Y -592.562,Z 488.458,A 0.000,B 0.000,C 90.000,E1 298.359} C_DIS
LIN {X -0.193,Y -594.405,Z 488.452,A 0.000,B 0.000,C 90.000,E1 297.334} C_DIS
LIN {X 0.247,Y -596.040,Z 488.446,A 0.000,B 0.000,C 90.000,E1 296.232} C_DIS
LIN {X -0.096,Y -597.435,Z 488.440,A 0.000,B 0.000,C 90.000,E1 295.207} C_DIS
LIN {X 0.198,Y -598.314,Z 488.436,A 0.000,B 0.000,C 90.000,E1 294.387} C_DIS
LIN {X 0.101,Y -599.524,Z 488.428,A 0.000,B 0.000,C 90.000,E1 293.078} C_DIS
LIN {X 0.022,Y -600.683,Z 488.421,A 0.000,B 0.000,C 90.000,E1 291.770} C_DIS
LIN {X -0.263,Y -601.668,Z 488.414,A 0.000,B 0.000,C 90.000,E1 290.482} C_DIS
LIN {X 0.120,Y -602.337,Z 488.408,A 0.000,B 0.000,C 90.000,E1 289.396} C_DIS
LIN {X 0.148,Y -603.153,Z 488.399,A 0.000,B 0.000,C 90.000,E1 287.819} C_DIS
LIN {X -0.200,Y -603.729,Z 488.393,A 0.000,B 0.000,C 90.000,E1 286.804} C_DIS
LIN {X -0.065,Y -604.334,Z 488.386,A 0.000,B 0.000,C 90.000,E1 285.481} C_DIS
LIN {X -0.092,Y -604.844,Z 488.379,A 0.000,B 0.000,C 90.000,E1 284.175} C_DIS
LIN {X -0.257,Y -605.151,Z 488.371,A 0.000,B 0.000,C 90.000,E1 282.883} C_DIS
LIN {X -0.148,Y -605.384,Z 488.366,A 0.000,B 0.000,C 90.000,E1 281.827} C_DIS
LIN {X -0.154,Y -605.536,Z 488.360,A 0.000,B 0.000,C 90.000,E1 280.782} C_DIS
LIN {X 0.178,Y -605.474,Z 488.353,A 0.000,B 0.000,C 90.000,E1 279.443} C_DIS
LIN {X -0.098,Y -605.260,Z 488.345,A 0.000,B 0.000,C 90.000,E1 278.163} C_DIS
LIN {X -0.185,Y -604.917,Z 488.340,A 0.000,B 0.000,C 90.000,E1 277.125} C_DIS
LIN {X -0.273,Y -604.443,Z 488.334,A 0.000,B 0.000,C 90.000,E1 276.087} C_DIS
LIN {X -0.070,Y -603.576,Z 488.326,A 0.000,B 0.000,C 90.000,E1 274.759} C_DIS
LIN {X -0.234,Y -602.720,Z 488.321,A 0.000,B 0.000,C 90.000,E1 273.726} C_DIS
LIN {X 0.195,Y -601.719,Z 488.315,A 0.000,B 0.000,C 90.000,E1 272.636} C_DIS
LIN {X -0.260,Y -600.767,Z 488.310,A 0.000,B 0.000,C 90.000,E1 271.892} C_DIS
LIN {X 0.137,Y -599.401,Z 488.305,A 0.000,B 0.000,C 90.000,E1 270.802} C_DIS
LIN {X 0.140,Y -597.517,Z 488.297,A 0.000,B 0.000,C 90.000,E1 269.484} C_DIS
LIN {X -0.122,Y -595.918,Z 488.291,A 0.000,B 0.000,C 90.000,E1 268.453} C_DIS
LIN {X 0.080,Y -593.406,Z 488.283,A 0.000,B 0.000,C 90.000,E1 266.846} C_DIS
LIN {X -0.007,Y -591.086,Z 488.275,A 0.000,B 0.000,C 90.000,E1 265.527} C_DIS
LIN {X -0.098,Y -588.557,Z 488.268,A 0.000,B 0.000,C 90.000,E1 264.204} C_DIS
LIN {X -0.167,Y -585.904,Z 488.260,A 0.000,B 0.000,C 90.000,E1 262.875} C_DIS
LIN {X 0.062,Y -583.808,Z 488.254,A 0.000,B 0.000,C 90.000,E1 261.781} C_DIS
LIN {X 0.227,Y -580.621,Z 488.245,A 0.000,B 0.000,C 90.000,E1 260.151} C_DIS
LIN {X -0.113,Y -578.390,Z 488.239,A 0.000,B 0.000,C 90.000,E1 259.106} C_DIS
LIN {X -0.157,Y -575.407,Z 488.232,A 0.000,B 0.000,C 90.000,E1 257.757} C_DIS
LIN {X -0.059,Y -571.759,Z 488.223,A 0.000,B 0.000,C 90.000,E1 256.117} C_DIS
LIN {X -0.091,Y -568.567,Z 488.215,A 0.000,B 0.000,C 90.000,E1 254.755} C_DIS
LIN {X -0.024,Y -565.214,Z 488.208,A 0.000,B 0.000,C 90.000,E1 253.378} C_DIS
LIN {X 0.064,Y -563.149,Z 488.203,A 0.000,B 0.000,C 90.000,E1 252.543} C_DIS
LIN {X 0.209,Y -559.546,Z 488.195,A 0.000,B 0.000,C 90.000,E1 251.148} C_DIS
LIN {X 0.291,Y -555.710,Z 488.188,A 0.000,B 0.000,C 90.000,E1 249.752} C_DIS
LIN {X -0.221,Y -551.649,Z 488.180,A 0.000,B 0.000,C 90.000,E1 248.411} C_DIS
LIN {X -0.148,Y -548.295,Z 488.174,A 0.000,B 0.000,C 90.000,E1 247.283} C_DIS
LIN {X -0.334,Y -544.778,Z 488.168,A 0.000,B 0.000,C 90.000,E1 246.177} C_DIS
LIN {X 0.102,Y -540.255,Z 488.160,A 0.000,B 0.000,C 90.000,E1 244.717} C_DIS
LIN {X -0.026,Y -535.607,Z 488.152,A 0.000,B 0.000,C 90.000,E1 243.307} C_DIS
LIN {X -0.237,Y -530.921,Z 488.144,A 0.000,B 0.000,C 90.000,E1 241.897} C_DIS
LIN {X 0.124,Y -525.289,Z 488.134,A 0.000,B 0.000,C 90.000,E1 240.127} C_DIS
LIN {X -0.101,Y -519.671,Z 488.124,A 0.000,B 0.000,C 90.000,E1 238.408} C_DIS
LIN {X -0.193,Y -515.891,Z 488.118,A 0.000,B 0.000,C 90.000,E1 237.248} C_DIS
LIN {X 0.023,Y -512.953,Z 488.113,A 0.000,B 0.000,C 90.000,E1 236.342} C_DIS
LIN {X 0.065,Y -506.945,Z 488.103,A 0.000,B 0.000,C 90.000,E1 234.562} C_DIS
LIN {X -0.214,Y -498.117,Z 488.088,A 0.000,B 0.000,C 90.000,E1 231.904} C_DIS
LIN {X -0.020,Y -492.722,Z 488.078,A 0.000,B 0.000,C 90.000,E1 230.070} C_DIS
LIN {X 0.159,Y -488.324,Z 488.070,A 0.000,B 0.000,C 90.000,E1 228.528} C_DIS
LIN {X 0.068,Y -483.218,Z 488.060,A 0.000,B 0.000,C 90.000,E1 226.701} C_DIS
LIN {X 0.171,Y -478.209,Z 488.049,A 0.000,B 0.000,C 90.000,E1 224.838} C_DIS
LIN {X -0.067,Y -472.653,Z 488.037,A 0.000,B 0.000,C 90.000,E1 222.690} C_DIS
LIN {X 0.168,Y -468.127,Z 488.027,A 0.000,B 0.000,C 90.000,E1 220.782} C_DIS
LIN {X 0.041,Y -463.102,Z 488.014,A 0.000,B 0.000,C 90.000,E1 218.588} C_DIS
LIN {X 0.188,Y -459.086,Z 488.004,A 0.000,B 0.000,C 90.000,E1 216.664} C_DIS
LIN {X -0.017,Y -455.220,Z 487.993,A 0.000,B 0.000,C 90.000,E1 214.771} C_DIS
LIN {X -0.222,Y -450.845,Z 487.981,A 0.000,B 0.000,C 90.000,E1 212.546} C_DIS
LIN {X -0.113,Y -447.260,Z 487.970,A 0.000,B 0.000,C 90.000,E1 210.590} C_DIS
LIN {X 0.066,Y -443.687,Z 487.959,A 0.000,B 0.000,C 90.000,E1 208.615} C_DIS
LIN {X -0.055,Y -440.189,Z 487.948,A 0.000,B 0.000,C 90.000,E1 206.668} C_DIS
LIN {X -0.067,Y -436.595,Z 487.937,A 0.000,B 0.000,C 90.000,E1 204.695} C_DIS
LIN {X -0.170,Y -434.254,Z 487.930,A 0.000,B 0.000,C 90.000,E1 203.387} C_DIS
LIN {X 0.131,Y -430.746,Z 487.919,A 0.000,B 0.000,C 90.000,E1 201.354} C_DIS
LIN {X 0.005,Y -426.970,Z 487.906,A 0.000,B 0.000,C 90.000,E1 199.033} C_DIS
LIN {X 0.035,Y -423.428,Z 487.893,A 0.000,B 0.000,C 90.000,E1 196.677} C_DIS
LIN {X -0.044,Y -420.664,Z 487.881,A 0.000,B 0.000,C 90.000,E1 194.662} C_DIS
LIN {X -0.132,Y -417.709,Z 487.868,A 0.000,B 0.000,C 90.000,E1 192.299} C_DIS
LIN {X -0.125,Y -415.310,Z 487.857,A 0.000,B 0.000,C 90.000,E1 190.254} C_DIS
LIN {X 0.194,Y -412.671,Z 487.844,A 0.000,B 0.000,C 90.000,E1 187.814} C_DIS
LIN {X -0.089,Y -410.350,Z 487.830,A 0.000,B 0.000,C 90.000,E1 185.448} C_DIS
LIN {X -0.124,Y -407.841,Z 487.815,A 0.000,B 0.000,C 90.000,E1 182.694} C_DIS
LIN {X 0.145,Y -405.837,Z 487.800,A 0.000,B 0.000,C 90.000,E1 179.885} C_DIS
LIN {X -0.054,Y -404.366,Z 487.784,A 0.000,B 0.000,C 90.000,E1 177.135} C_DIS
LIN {X 0.120,Y -403.346,Z 487.763,A 0.000,B 0.000,C 90.000,E1 173.280} C_DIS
LIN {X 0.066,Y -403.428,Z 487.743,A 0.000,B 0.000,C 90.000,E1 169.803} C_DIS
LIN {X 0.144,Y -404.011,Z 487.730,A 0.000,B 0.000,C 90.000,E1 167.353} C_DIS
LIN {X 0.020,Y -404.757,Z 487.718,A 0.000,B 0.000,C 90.000,E1 165.283} C_DIS
LIN {X -0.078,Y -405.615,Z 487.709,A 0.000,B 0.000,C 90.000,E1 163.559} C_DIS
LIN {X 0.066,Y -406.815,Z 487.697,A 0.000,B 0.000,C 90.000,E1 161.456} C_DIS
LIN {X 0.098,Y -408.645,Z 487.684,A 0.000,B 0.000,C 90.000,E1 159.028} C_DIS
LIN {X -0.168,Y -411.111,Z 487.668,A 0.000,B 0.000,C 90.000,E1 156.305} C_DIS
LIN {X -0.148,Y -413.446,Z 487.655,A 0.000,B 0.000,C 90.000,E1 153.896} C_DIS
LIN {X 0.008,Y -415.591,Z 487.643,A 0.000,B 0.000,C 90.000,E1 151.820} C_DIS
LIN {X -0.148,Y -417.609,Z 487.632,A 0.000,B 0.000,C 90.000,E1 149.793} C_DIS
LIN {X 0.125,Y -419.951,Z 487.619,A 0.000,B 0.000,C 90.000,E1 147.375} C_DIS
LIN {X -0.221,Y -421.860,Z 487.608,A 0.000,B 0.000,C 90.000,E1 145.388} C_DIS
LIN {X -0.257,Y -423.458,Z 487.598,A 0.000,B 0.000,C 90.000,E1 143.703} C_DIS
LIN {X -0.013,Y -425.129,Z 487.589,A 0.000,B 0.000,C 90.000,E1 141.984} C_DIS
LIN {X -0.034,Y -426.437,Z 487.581,A 0.000,B 0.000,C 90.000,E1 140.642} C_DIS
LIN {X -0.031,Y -427.744,Z 487.574,A 0.000,B 0.000,C 90.000,E1 139.299} C_DIS
LIN {X -0.017,Y -428.894,Z 487.566,A 0.000,B 0.000,C 90.000,E1 137.957} C_DIS
LIN {X -0.020,Y -429.848,Z 487.559,A 0.000,B 0.000,C 90.000,E1 136.620} C_DIS
LIN {X -0.008,Y -430.633,Z 487.552,A 0.000,B 0.000,C 90.000,E1 135.283} C_DIS
LIN {X 0.015,Y -431.114,Z 487.544,A 0.000,B 0.000,C 90.000,E1 133.947} C_DIS
LIN {X 0.120,Y -431.331,Z 487.539,A 0.000,B 0.000,C 90.000,E1 132.933} C_DIS
LIN {X 0.156,Y -431.143,Z 487.531,A 0.000,B 0.000,C 90.000,E1 131.595} C_DIS
LIN {X -0.025,Y -430.655,Z 487.526,A 0.000,B 0.000,C 90.000,E1 130.620} C_DIS
LIN {X -0.211,Y -429.899,Z 487.520,A 0.000,B 0.000,C 90.000,E1 129.644} C_DIS
LIN {X -0.163,Y -428.512,Z 487.513,A 0.000,B 0.000,C 90.000,E1 128.302} C_DIS
LIN {X -0.044,Y -427.365,Z 487.507,A 0.000,B 0.000,C 90.000,E1 127.282} C_DIS
LIN {X 0.169,Y -426.527,Z 487.503,A 0.000,B 0.000,C 90.000,E1 126.583} C_DIS
LIN {X -0.138,Y -424.075,Z 487.494,A 0.000,B 0.000,C 90.000,E1 124.945} C_DIS
LIN {X 0.037,Y -421.737,Z 487.486,A 0.000,B 0.000,C 90.000,E1 123.420} C_DIS
LIN {X -0.002,Y -421.737,Z 487.486,A 0.000,B 0.000,C 90.000,E1 123.420} C_DIS
LIN {X 0.042,Y -430.949,Z 487.468,A 0.000,B 0.000,C 90.000,E1 120.207} C_DIS
LIN {X -0.009,Y -440.007,Z 487.448,A 0.000,B 0.000,C 90.000,E1 116.565} C_DIS
LIN {X 0.186,Y -444.796,Z 487.439,A 0.000,B 0.000,C 90.000,E1 114.899} C_DIS
LIN {X -0.140,Y -453.902,Z 487.417,A 0.000,B 0.000,C 90.000,E1 111.046} C_DIS
LIN {X -0.125,Y -457.394,Z 487.410,A 0.000,B 0.000,C 90.000,E1 109.758} C_DIS
LIN {X -0.041,Y -466.033,Z 487.387,A 0.000,B 0.000,C 90.000,E1 105.607} C_DIS
LIN {X 0.133,Y -467.600,Z 487.383,A 0.000,B 0.000,C 90.000,E1 104.954} C_DIS
LIN {X -0.254,Y -468.436,Z 487.380,A 0.000,B 0.000,C 90.000,E1 104.481} C_DIS
LIN {X 0.159,Y -469.032,Z 487.380,A 0.000,B 0.000,C 90.000,E1 104.426} C_DIS
LIN {X 0.054,Y -480.154,Z 487.380,A 0.000,B 0.000,C 90.000,E1 104.356} C_DIS
LIN {X -0.034,Y -486.045,Z 487.379,A 0.000,B 0.000,C 90.000,E1 104.300} C_DIS
LIN {X 0.127,Y -500.900,Z 487.378,A 0.000,B 0.000,C 90.000,E1 104.064} C_DIS
LIN {X 0.058,Y -507.486,Z 487.378,A 0.000,B 0.000,C 90.000,E1 103.953} C_DIS
LIN {X -0.162,Y -514.621,Z 487.377,A 0.000,B 0.000,C 90.000,E1 103.828} C_DIS
LIN {X -0.006,Y -528.163,Z 487.375,A 0.000,B 0.000,C 90.000,E1 103.480} C_DIS
LIN {X 0.220,Y -538.723,Z 487.373,A 0.000,B 0.000,C 90.000,E1 103.175} C_DIS
LIN {X -0.057,Y -545.299,Z 487.372,A 0.000,B 0.000,C 90.000,E1 103.008} C_DIS
LIN {X 0.111,Y -555.417,Z 487.370,A 0.000,B 0.000,C 90.000,E1 102.647} C_DIS
LIN {X -0.065,Y -561.685,Z 487.369,A 0.000,B 0.000,C 90.000,E1 102.411} C_DIS
LIN {X -0.039,Y -568.225,Z 487.367,A 0.000,B 0.000,C 90.000,E1 102.119} C_DIS
LIN {X -0.219,Y -574.632,Z 487.366,A 0.000,B 0.000,C 90.000,E1 101.827} C_DIS
LIN {X -0.058,Y -580.708,Z 487.364,A 0.000,B 0.000,C 90.000,E1 101.478} C_DIS
LIN {X 0.109,Y -585.584,Z 487.362,A 0.000,B 0.000,C 90.000,E1 101.186} C_DIS
LIN {X 0.074,Y -593.134,Z 487.360,A 0.000,B 0.000,C 90.000,E1 100.715} C_DIS
LIN {X 0.069,Y -598.953,Z 487.357,A 0.000,B 0.000,C 90.000,E1 100.310} C_DIS
LIN {X -0.217,Y -604.561,Z 487.355,A 0.000,B 0.000,C 90.000,E1 99.905} C_DIS
LIN {X 0.159,Y -609.612,Z 487.353,A 0.000,B 0.000,C 90.000,E1 99.443} C_DIS
LIN {X 0.232,Y -615.858,Z 487.349,A 0.000,B 0.000,C 90.000,E1 98.859} C_DIS
LIN {X -0.258,Y -621.919,Z 487.346,A 0.000,B 0.000,C 90.000,E1 98.276} C_DIS
LIN {X -0.090,Y -628.062,Z 487.342,A 0.000,B 0.000,C 90.000,E1 97.530} C_DIS
LIN {X -0.044,Y -632.901,Z 487.338,A 0.000,B 0.000,C 90.000,E1 96.891} C_DIS
LIN {X -0.169,Y -637.917,Z 487.334,A 0.000,B 0.000,C 90.000,E1 96.144} C_DIS
LIN {X -0.178,Y -642.298,Z 487.330,A 0.000,B 0.000,C 90.000,E1 95.391} C_DIS
LIN {X -0.091,Y -645.614,Z 487.326,A 0.000,B 0.000,C 90.000,E1 94.759} C_DIS
LIN {X -0.090,Y -649.171,Z 487.322,A 0.000,B 0.000,C 90.000,E1 94.012} C_DIS
LIN {X 0.116,Y -651.287,Z 487.320,A 0.000,B 0.000,C 90.000,E1 93.498} C_DIS
LIN {X -0.273,Y -653.152,Z 487.317,A 0.000,B 0.000,C 90.000,E1 93.037} C_DIS
LIN {X -0.034,Y -654.677,Z 487.314,A 0.000,B 0.000,C 90.000,E1 92.522} C_DIS
LIN {X 0.223,Y -655.904,Z 487.311,A 0.000,B 0.000,C 90.000,E1 92.007} C_DIS
LIN {X 0.048,Y -656.498,Z 487.310,A 0.000,B 0.000,C 90.000,E1 91.776} C_DIS
LIN {X 0.317,Y -657.411,Z 487.307,A 0.000,B 0.000,C 90.000,E1 91.260} C_DIS
LIN {X -0.252,Y -658.188,Z 487.303,A 0.000,B 0.000,C 90.000,E1 90.573} C_DIS
LIN {X 0.034,Y -658.453,Z 487.300,A 0.000,B 0.000,C 90.000,E1 90.057} C_DIS
LIN {X 0.321,Y -658.370,Z 487.298,A 0.000,B 0.000,C 90.000,E1 89.542} C_DIS
LIN {X -0.238,Y -657.811,Z 487.294,A 0.000,B 0.000,C 90.000,E1 88.854} C_DIS
LIN {X 0.043,Y -657.263,Z 487.291,A 0.000,B 0.000,C 90.000,E1 88.339} C_DIS
LIN {X -0.316,Y -656.344,Z 487.288,A 0.000,B 0.000,C 90.000,E1 87.879} C_DIS
LIN {X -0.045,Y -655.204,Z 487.285,A 0.000,B 0.000,C 90.000,E1 87.364} C_DIS
LIN {X 0.212,Y -653.771,Z 487.283,A 0.000,B 0.000,C 90.000,E1 86.849} C_DIS
LIN {X -0.155,Y -652.086,Z 487.280,A 0.000,B 0.000,C 90.000,E1 86.388} C_DIS
LIN {X -0.091,Y -649.097,Z 487.276,A 0.000,B 0.000,C 90.000,E1 85.641} C_DIS
LIN {X 0.057,Y -646.195,Z 487.272,A 0.000,B 0.000,C 90.000,E1 85.008} C_DIS
LIN {X 0.177,Y -642.841,Z 487.269,A 0.000,B 0.000,C 90.000,E1 84.375} C_DIS
LIN {X 0.264,Y -639.091,Z 487.265,A 0.000,B 0.000,C 90.000,E1 83.742} C_DIS
LIN {X 0.182,Y -634.061,Z 487.261,A 0.000,B 0.000,C 90.000,E1 82.996} C_DIS
LIN {X 0.124,Y -628.354,Z 487.257,A 0.000,B 0.000,C 90.000,E1 82.243} C_DIS
LIN {X 0.234,Y -624.123,Z 487.254,A 0.000,B 0.000,C 90.000,E1 81.724} C_DIS
LIN {X -0.142,Y -620.848,Z 487.252,A 0.000,B 0.000,C 90.000,E1 81.376} C_DIS
LIN {X 0.090,Y -616.251,Z 487.249,A 0.000,B 0.000,C 90.000,E1 80.849} C_DIS
LIN {X 0.177,Y -609.960,Z 487.246,A 0.000,B 0.000,C 90.000,E1 80.208} C_DIS
LIN {X -0.257,Y -603.430,Z 487.242,A 0.000,B 0.000,C 90.000,E1 79.634} C_DIS
LIN {X 0.233,Y -597.977,Z 487.240,A 0.000,B 0.000,C 90.000,E1 79.106} C_DIS
LIN {X 0.256,Y -593.740,Z 487.238,A 0.000,B 0.000,C 90.000,E1 78.757} C_DIS
LIN {X 0.018,Y -587.763,Z 487.235,A 0.000,B 0.000,C 90.000,E1 78.342} C_DIS
LIN {X -0.002,Y -581.449,Z 487.233,A 0.000,B 0.000,C 90.000,E1 77.937} C_DIS
LIN {X 0.086,Y -576.506,Z 487.231,A 0.000,B 0.000,C 90.000,E1 77.645} C_DIS
LIN {X 0.092,Y -569.723,Z 487.230,A 0.000,B 0.000,C 90.000,E1 77.297} C_DIS
LIN {X 0.150,Y -562.189,Z 487.228,A 0.000,B 0.000,C 90.000,E1 76.992} C_DIS
LIN {X -0.110,Y -555.936,Z 487.227,A 0.000,B 0.000,C 90.000,E1 76.825} C_DIS
LIN {X 0.087,Y -552.101,Z 487.226,A 0.000,B 0.000,C 90.000,E1 76.700} C_DIS
LIN {X 0.186,Y -543.677,Z 487.225,A 0.000,B 0.000,C 90.000,E1 76.533} C_DIS
LIN {X 0.269,Y -539.500,Z 487.225,A 0.000,B 0.000,C 90.000,E1 76.464} C_DIS
LIN {X 0.178,Y -529.143,Z 487.225,A 0.000,B 0.000,C 90.000,E1 76.408} C_DIS
LIN {X 0.027,Y -523.025,Z 487.225,A 0.000,B 0.000,C 90.000,E1 76.408} C_DIS
LIN {X -0.017,Y -479.800,Z 487.225,A 0.000,B 0.000,C 90.000,E1 76.408} C_DIS
LIN {X -0.054,Y -474.119,Z 487.200,A 0.000,B 0.000,C 90.000,E1 72.054} C_DIS
LIN {X -0.186,Y -465.582,Z 487.172,A 0.000,B 0.000,C 90.000,E1 67.050} C_DIS
LIN {X 0.201,Y -457.122,Z 487.149,A 0.000,B 0.000,C 90.000,E1 62.871} C_DIS
LIN {X -0.092,Y -455.540,Z 487.144,A 0.000,B 0.000,C 90.000,E1 61.948} C_DIS
LIN {X 0.119,Y -452.613,Z 487.137,A 0.000,B 0.000,C 90.000,E1 60.717} C_DIS
LIN {X 0.078,Y -452.607,Z 487.137,A 0.000,B 0.000,C 90.000,E1 60.717} C_DIS
LIN {X -0.083,Y -459.106,Z 487.131,A 0.000,B 0.000,C 90.000,E1 59.537} C_DIS
LIN {X -0.097,Y -463.209,Z 487.126,A 0.000,B 0.000,C 90.000,E1 58.742} C_DIS
LIN {X 0.176,Y -466.262,Z 487.123,A 0.000,B 0.000,C 90.000,E1 58.074} C_DIS
LIN {X 0.079,Y -469.089,Z 487.119,A 0.000,B 0.000,C 90.000,E1 57.454} C_DIS
LIN {X 0.004,Y -471.632,Z 487.116,A 0.000,B 0.000,C 90.000,E1 56.834} C_DIS
LIN {X -0.053,Y -473.788,Z 487.112,A 0.000,B 0.000,C 90.000,E1 56.215} C_DIS
LIN {X 0.083,Y -476.615,Z 487.107,A 0.000,B 0.000,C 90.000,E1 55.261} C_DIS
LIN {X 0.059,Y -478.142,Z 487.104,A 0.000,B 0.000,C 90.000,E1 54.642} C_DIS
LIN {X 0.129,Y -479.949,Z 487.098,A 0.000,B 0.000,C 90.000,E1 53.703} C_DIS
LIN {X 0.225,Y -481.430,Z 487.093,A 0.000,B 0.000,C 90.000,E1 52.763} C_DIS
LIN {X 0.042,Y -482.542,Z 487.088,A 0.000,B 0.000,C 90.000,E1 51.859} C_DIS
LIN {X 0.091,Y -483.451,Z 487.083,A 0.000,B 0.000,C 90.000,E1 50.928} C_DIS
LIN {X 0.224,Y -484.091,Z 487.078,A 0.000,B 0.000,C 90.000,E1 49.989} C_DIS
LIN {X -0.060,Y -484.988,Z 487.069,A 0.000,B 0.000,C 90.000,E1 48.485} C_DIS
LIN {X 0.176,Y -485.403,Z 487.063,A 0.000,B 0.000,C 90.000,E1 47.229} C_DIS
LIN {X -0.266,Y -485.539,Z 487.056,A 0.000,B 0.000,C 90.000,E1 46.053} C_DIS
LIN {X -0.027,Y -485.569,Z 487.049,A 0.000,B 0.000,C 90.000,E1 44.798} C_DIS
LIN {X 0.214,Y -485.329,Z 487.042,A 0.000,B 0.000,C 90.000,E1 43.542} C_DIS
LIN {X 0.312,Y -485.039,Z 487.037,A 0.000,B 0.000,C 90.000,E1 42.609} C_DIS
LIN {X -0.324,Y -484.268,Z 487.028,A 0.000,B 0.000,C 90.000,E1 41.148} C_DIS
LIN {X -0.110,Y -483.133,Z 487.018,A 0.000,B 0.000,C 90.000,E1 39.277} C_DIS
LIN {X -0.228,Y -481.990,Z 487.008,A 0.000,B 0.000,C 90.000,E1 37.443} C_DIS
LIN {X -0.095,Y -480.926,Z 486.999,A 0.000,B 0.000,C 90.000,E1 35.884} C_DIS
LIN {X 0.216,Y -479.303,Z 486.989,A 0.000,B 0.000,C 90.000,E1 33.992} C_DIS
LIN {X 0.220,Y -478.165,Z 486.982,A 0.000,B 0.000,C 90.000,E1 32.752} C_DIS
LIN {X 0.146,Y -476.655,Z 486.974,A 0.000,B 0.000,C 90.000,E1 31.209} C_DIS
LIN {X 0.226,Y -474.692,Z 486.963,A 0.000,B 0.000,C 90.000,E1 29.333} C_DIS
LIN {X -0.207,Y -472.669,Z 486.953,A 0.000,B 0.000,C 90.000,E1 27.513} C_DIS
LIN {X -0.005,Y -471.124,Z 486.944,A 0.000,B 0.000,C 90.000,E1 25.924} C_DIS
LIN {X 0.124,Y -469.426,Z 486.934,A 0.000,B 0.000,C 90.000,E1 24.027} C_DIS
LIN {X -0.082,Y -467.626,Z 486.920,A 0.000,B 0.000,C 90.000,E1 21.535} C_DIS
LIN {X -0.094,Y -466.174,Z 486.906,A 0.000,B 0.000,C 90.000,E1 19.014} C_DIS
LIN {X -0.100,Y -465.029,Z 486.893,A 0.000,B 0.000,C 90.000,E1 16.804} C_DIS
LIN {X 0.027,Y -463.810,Z 486.878,A 0.000,B 0.000,C 90.000,E1 13.939} C_DIS
LIN {X -0.079,Y -463.018,Z 486.860,A 0.000,B 0.000,C 90.000,E1 10.782} C_DIS
LIN {X -0.159,Y -462.964,Z 486.844,A 0.000,B 0.000,C 90.000,E1 7.936} C_DIS
LIN {X 0.082,Y -463.724,Z 486.825,A 0.000,B 0.000,C 90.000,E1 4.416} C_DIS
LIN {X 0.004,Y -464.999,Z 486.811,A 0.000,B 0.000,C 90.000,E1 1.892} C_DIS
LIN {X -0.069,Y -467.371,Z 486.794,A 0.000,B 0.000,C 90.000,E1 358.854} C_DIS
LIN {X 0.004,Y -470.570,Z 486.776,A 0.000,B 0.000,C 90.000,E1 355.698} C_DIS
LIN {X -0.133,Y -472.477,Z 486.767,A 0.000,B 0.000,C 90.000,E1 354.147} C_DIS
LIN {X -0.061,Y -475.352,Z 486.755,A 0.000,B 0.000,C 90.000,E1 351.951} C_DIS
LIN {X 0.009,Y -478.909,Z 486.741,A 0.000,B 0.000,C 90.000,E1 349.454} C_DIS
LIN {X -0.052,Y -485.322,Z 486.721,A 0.000,B 0.000,C 90.000,E1 345.755} C_DIS
LIN {X -0.082,Y -489.774,Z 486.709,A 0.000,B 0.000,C 90.000,E1 343.614} C_DIS
LIN {X 0.186,Y -495.144,Z 486.695,A 0.000,B 0.000,C 90.000,E1 341.148} C_DIS
LIN {X -0.233,Y -499.972,Z 486.684,A 0.000,B 0.000,C 90.000,E1 339.082} C_DIS
LIN {X 0.129,Y -503.401,Z 486.675,A 0.000,B 0.000,C 90.000,E1 337.539} C_DIS
LIN {X -0.191,Y -508.033,Z 486.664,A 0.000,B 0.000,C 90.000,E1 335.485} C_DIS
LIN {X 0.053,Y -511.265,Z 486.655,A 0.000,B 0.000,C 90.000,E1 333.973} C_DIS
LIN {X -0.223,Y -515.098,Z 486.646,A 0.000,B 0.000,C 90.000,E1 332.231} C_DIS
LIN {X 0.171,Y -518.344,Z 486.637,A 0.000,B 0.000,C 90.000,E1 330.717} C_DIS
LIN {X 0.241,Y -523.075,Z 486.626,A 0.000,B 0.000,C 90.000,E1 328.663} C_DIS
LIN {X -0.112,Y -526.511,Z 486.618,A 0.000,B 0.000,C 90.000,E1 327.248} C_DIS
LIN {X -0.141,Y -530.683,Z 486.608,A 0.000,B 0.000,C 90.000,E1 325.515} C_DIS
LIN {X -0.069,Y -533.518,Z 486.602,A 0.000,B 0.000,C 90.000,E1 324.356} C_DIS
LIN {X -0.085,Y -536.348,Z 486.596,A 0.000,B 0.000,C 90.000,E1 323.210} C_DIS
LIN {X 0.304,Y -540.580,Z 486.586,A 0.000,B 0.000,C 90.000,E1 321.457} C_DIS
LIN {X 0.021,Y -544.786,Z 486.577,A 0.000,B 0.000,C 90.000,E1 319.784} C_DIS
LIN {X -0.288,Y -548.233,Z 486.569,A 0.000,B 0.000,C 90.000,E1 318.405} C_DIS
LIN {X -0.120,Y -552.259,Z 486.559,A 0.000,B 0.000,C 90.000,E1 316.701} C_DIS
LIN {X 0.075,Y -555.488,Z 486.552,A 0.000,B 0.000,C 90.000,E1 315.283} C_DIS
LIN {X -0.121,Y -558.074,Z 486.545,A 0.000,B 0.000,C 90.000,E1 314.190} C_DIS
LIN {X -0.144,Y -561.925,Z 486.536,A 0.000,B 0.000,C 90.000,E1 312.528} C_DIS
LIN {X -0.148,Y -565.114,Z 486.529,A 0.000,B 0.000,C 90.000,E1 311.148} C_DIS
LIN {X -0.101,Y -568.190,Z 486.521,A 0.000,B 0.000,C 90.000,E1 309.769} C_DIS
LIN {X 0.074,Y -571.360,Z 486.513,A 0.000,B 0.000,C 90.000,E1 308.382} C_DIS
LIN {X -0.039,Y -574.511,Z 486.506,A 0.000,B 0.000,C 90.000,E1 307.030} C_DIS
LIN {X 0.226,Y -579.009,Z 486.495,A 0.000,B 0.000,C 90.000,E1 305.105} C_DIS
LIN {X 0.085,Y -582.910,Z 486.486,A 0.000,B 0.000,C 90.000,E1 303.499} C_DIS
LIN {X 0.322,Y -586.148,Z 486.479,A 0.000,B 0.000,C 90.000,E1 302.133} C_DIS
LIN {X 0.123,Y -588.499,Z 486.473,A 0.000,B 0.000,C 90.000,E1 301.082} C_DIS
LIN {X 0.153,Y -591.265,Z 486.465,A 0.000,B 0.000,C 90.000,E1 299.745} C_DIS
LIN {X -0.066,Y -593.770,Z 486.458,A 0.000,B 0.000,C 90.000,E1 298.437} C_DIS
LIN {X -0.159,Y -595.668,Z 486.452,A 0.000,B 0.000,C 90.000,E1 297.385} C_DIS
LIN {X -0.052,Y -597.728,Z 486.445,A 0.000,B 0.000,C 90.000,E1 296.052} C_DIS
LIN {X 0.174,Y -599.063,Z 486.439,A 0.000,B 0.000,C 90.000,E1 294.975} C_DIS
LIN {X -0.131,Y -600.163,Z 486.433,A 0.000,B 0.000,C 90.000,E1 293.951} C_DIS
LIN {X 0.283,Y -601.653,Z 486.424,A 0.000,B 0.000,C 90.000,E1 292.333} C_DIS
LIN {X 0.314,Y -602.564,Z 486.418,A 0.000,B 0.000,C 90.000,E1 291.280} C_DIS
LIN {X 0.061,Y -603.576,Z 486.411,A 0.000,B 0.000,C 90.000,E1 289.993} C_DIS
